  MoveL 8467 to (-32, -51.45, -12.28) mm, rotated rx 180 ry 0 rz 90 deg; joints [71.833, -17.532, 85.378, 0, 22.154, 71.833]
  MoveL 8468 to (-30.9, -50.4, -12.69) mm, rotated rx 180 ry 0 rz 90 deg; joints [71.879, -17.498, 85.311, 0, 22.187, 71.879]
  MoveL 8469 to (-30.06, -49.13, -13.09) mm, rotated rx 180 ry 0 rz 90 deg; joints [71.929, -17.47, 85.268, 0, 22.202, 71.929]
  MoveL 8470 to (-29.55, -47.71, -13.5) mm, rotated rx 180 ry 0 rz 90 deg; joints [71.98, -17.448, 85.251, 0, 22.197, 71.98]
  MoveL 8471 to (-25.22, -30.8, -13.5) mm, rotated rx 180 ry 0 rz 90 deg; joints [72.572, -17.467, 85.325, 0, 22.141, 72.572]
  MoveL 8472 to (-24.37, -27.48, -13.5) mm, rotated rx 180 ry 0 rz 90 deg; joints [72.688, -17.47, 85.338, 0, 22.131, 72.688]
  MoveL 8473 to (-24.29, -27.01, -13.5) mm, rotated rx 180 ry 0 rz 90 deg; joints [72.704, -17.471, 85.343, 0, 22.128, 72.704]
  MoveC 8474 to (-25.15, -24.96, -13.5) mm, rotated rx -180 ry 0 rz 90 deg; joints [72.762, -17.497, 85.447, 0, 22.05, 72.762] to (-27.01, -23.75, -13.5) mm, rotated rx -180 ry 0 rz 90 deg; joints [72.782, -17.536, 85.602, 0, 21.933, 72.782]
  MoveC 8475 to (-27.34, -23.73, -13.5) mm, rotated rx 180 ry 0 rz 90 deg; joints [72.78, -17.542, 85.626, 0, 21.916, 72.78] to (-27.66, -23.77, -13.5) mm, rotated rx -180 ry 0 rz 90 deg; joints [72.775, -17.547, 85.647, 0, 21.9, 72.775]
  MoveL 8476 to (-34.52, -25.11, -13.5) mm, rotated rx 180 ry 0 rz 90 deg; joints [72.662, -17.657, 86.093, 0, 21.564, 72.662]
  MoveL 8477 to (-63.97, -30.99, -13.5) mm, rotated rx 180 ry 0 rz 90 deg; joints [72.162, -18.107, 87.975, 0, 20.132, 72.162]
  MoveL 8478 to (-68.88, -32, -13.5) mm, rotated rx 180 ry 0 rz 90 deg; joints [72.076, -18.178, 88.284, 0, 19.894, 72.076]
  MoveC 8479 to (-70.35, -32.85, -13.5) mm, rotated rx -180 ry 0 rz 90 deg; joints [72.032, -18.197, 88.364, 0, 19.832, 72.032] to (-71.01, -34.41, -13.5) mm, rotated rx -180 ry 0 rz 90 deg; joints [71.974, -18.199, 88.375, 0, 19.824, 71.974]
  MoveC 8480 to (-71.02, -34.67, -13.5) mm, rotated rx -180 ry 0 rz 90 deg; joints [71.965, -18.198, 88.37, 0, 19.828, 71.965] to (-71.03, -34.93, -13.5) mm, rotated rx 180 ry 0 rz 90 deg; joints [71.956, -18.197, 88.365, 0, 19.832, 71.956]
  MoveL 8481 to (-71.03, -68.06, -13.5) mm, rotated rx 180 ry 0 rz 90 deg; joints [70.866, -18.023, 87.616, 0, 20.407, 70.866]
  MoveC 8482 to (-70.26, -69.94, -13.5) mm, rotated rx -180 ry 0 rz 90 deg; joints [70.813, -18.001, 87.521, 0, 20.48, 70.813] to (-68.4, -70.75, -13.5) mm, rotated rx 180 ry 0 rz 90 deg; joints [70.808, -17.967, 87.377, 0, 20.59, 70.808]
  MoveC 8483 to (-67.86, -70.75, -13.5) mm, rotated rx 180 ry 0 rz 90 deg; joints [70.814, -17.958, 87.34, 0, 20.618, 70.814] to (-67.31, -70.75, -13.5) mm, rotated rx 180 ry 0 rz 90 deg; joints [70.82, -17.949, 87.303, 0, 20.646, 70.82]
  MoveC 8484 to (-52.36, -70.49, -13.5) mm, rotated rx 180 ry 0 rz 90 deg; joints [70.997, -17.707, 86.295, 0, 21.412, 70.997] to (-37.4, -70.16, -13.5) mm, rotated rx 180 ry 0 rz 90 deg; joints [71.173, -17.454, 85.277, 0, 22.178, 71.173]
  MoveC 8485 to (-35.88, -69.65, -13.5) mm, rotated rx 180 ry 0 rz 90 deg; joints [71.205, -17.431, 85.183, 0, 22.248, 71.205] to (-34.9, -68.38, -13.5) mm, rotated rx 180 ry 0 rz 90 deg; joints [71.257, -17.421, 85.146, 0, 22.276, 71.257]
  MoveC 8486 to (-34.73, -67.86, -13.5) mm, rotated rx 180 ry 0 rz 90 deg; joints [71.275, -17.421, 85.146, 0, 22.276, 71.275] to (-34.59, -67.34, -13.5) mm, rotated rx 180 ry 0 rz 90 deg; joints [71.294, -17.422, 85.148, 0, 22.274, 71.294]
  MoveL 8487 to (-29.55, -47.71, -13.5) mm, rotated rx 180 ry 0 rz 90 deg; joints [71.98, -17.448, 85.251, 0, 22.197, 71.98]
  MoveL 8488 to (-36.87, -45.83, -13.5) mm, rotated rx 180 ry 0 rz 90 deg; joints [71.964, -17.585, 85.799, 0, 21.786, 71.964]
  MoveL 8489 to (-36.87, -45.83, -10.5) mm, rotated rx 180 ry 0 rz 90 deg; joints [71.964, -17.739, 85.902, 0, 21.838, 71.964]
  Establecer velocidad (1000.0 mm/s)
  MoveL 8490 to (-36.87, -45.83, 10) mm, rotated rx 180 ry 0 rz 90 deg; joints [71.964, -18.794, 86.589, 0, 22.206, 71.964]
  Establecer velocidad (66.7 mm/s)
  MoveL 8491 to (5.19, -66.61, 10) mm, rotated rx 180 ry 0 rz 90 deg; joints [71.74, -17.89, 83.159, 0, 24.731, 71.74]
  MoveL 8492 to (5.19, -66.61, -10.5) mm, rotated rx 180 ry 0 rz 90 deg; joints [71.74, -16.849, 82.47, 0, 24.38, 71.74]
  MoveL 8493 to (6.49, -67.39, -10.91) mm, rotated rx 180 ry 0 rz 90 deg; joints [71.729, -16.798, 82.344, 0, 24.454, 71.729]
  MoveL 8494 to (7.96, -67.76, -11.31) mm, rotated rx -180 ry 0 rz 90 deg; joints [71.733, -16.747, 82.216, 0, 24.531, 71.733]
  MoveL 8495 to (9.48, -67.7, -11.72) mm, rotated rx -180 ry 0 rz 90 deg; joints [71.75, -16.697, 82.094, 0, 24.602, 71.75]
  MoveL 8496 to (10.92, -67.23, -12.13) mm, rotated rx -180 ry 0 rz 90 deg; joints [71.78, -16.651, 81.988, 0, 24.663, 71.78]
  MoveL 8497 to (12.18, -66.38, -12.53) mm, rotated rx -180 ry 0 rz 90 deg; joints [71.82, -16.611, 81.903, 0, 24.708, 71.82]
  MoveL 8498 to (13.16, -65.21, -12.94) mm, rotated rx 180 ry 0 rz 90 deg; joints [71.866, -16.579, 81.847, 0, 24.732, 71.866]
  MoveL 8499 to (13.78, -63.83, -13.34) mm, rotated rx 180 ry 0 rz 90 deg; joints [71.916, -16.555, 81.821, 0, 24.734, 71.916]
  MoveL 8500 to (13.96, -62.32, -13.75) mm, rotated rx 180 ry 0 rz 90 deg; joints [71.966, -16.541, 81.829, 0, 24.711, 71.966]
  MoveL 8501 to (13.96, -51.49, -13.75) mm, rotated rx -180 ry 0 rz 90 deg; joints [72.307, -16.609, 82.081, 0, 24.528, 72.307]
  MoveL 8502 to (13.96, -34.43, -13.75) mm, rotated rx 180 ry 0 rz 90 deg; joints [72.846, -16.713, 82.466, 0, 24.247, 72.846]
  MoveC 8503 to (11.96, -34.42, -13.75) mm, rotated rx 180 ry 0 rz 90 deg; joints [72.827, -16.752, 82.61, 0, 24.141, 72.827] to (10.29, -35.54, -13.75) mm, rotated rx 180 ry 0 rz 90 deg; joints [72.775, -16.777, 82.704, 0, 24.072, 72.775]
  MoveL 8504 to (10, -36.48, -13.75) mm, rotated rx 180 ry 0 rz 90 deg; joints [72.742, -16.777, 82.705, 0, 24.072, 72.742]
  MoveL 8505 to (2.17, -64.91, -13.75) mm, rotated rx -180 ry 0 rz 90 deg; joints [71.762, -16.753, 82.614, 0, 24.139, 71.762]
  MoveL 8506 to (1.94, -65.86, -13.75) mm, rotated rx -180 ry 0 rz 90 deg; joints [71.73, -16.751, 82.608, 0, 24.143, 71.73]
  MoveC 8507 to (2.52, -67.83, -13.75) mm, rotated rx 180 ry 0 rz 90 deg; joints [71.674, -16.727, 82.52, 0, 24.207, 71.674] to (4.26, -68.91, -13.75) mm, rotated rx 180 ry 0 rz 90 deg; joints [71.658, -16.687, 82.37, 0, 24.317, 71.658]
  MoveL 8508 to (5.21, -68.93, -13.75) mm, rotated rx 180 ry 0 rz 90 deg; joints [71.667, -16.669, 82.301, 0, 24.367, 71.667]
  MoveL 8509 to (13.96, -68.54, -13.75) mm, rotated rx -180 ry 0 rz 90 deg; joints [71.77, -16.501, 81.683, 0, 24.818, 71.77]
  MoveL 8510 to (13.96, -51.49, -13.75) mm, rotated rx -180 ry 0 rz 90 deg; joints [72.307, -16.609, 82.081, 0, 24.528, 72.307]
  MoveL 8511 to (6.41, -51.49, -13.75) mm, rotated rx 180 ry 0 rz 90 deg; joints [72.23, -16.755, 82.623, 0, 24.132, 72.23]
  MoveL 8512 to (6.41, -51.49, -10.75) mm, rotated rx -180 ry 0 rz 90 deg; joints [72.23, -16.908, 82.726, 0, 24.182, 72.23]
  Establecer velocidad (1000.0 mm/s)
  MoveL 8513 to (6.41, -51.49, 10) mm, rotated rx 180 ry 0 rz 90 deg; joints [72.23, -17.962, 83.423, 0, 24.539, 72.23]
  Establecer velocidad (66.7 mm/s)
  MoveL 8514 to (-39.34, -52.07, 10) mm, rotated rx -180 ry 0 rz 90 deg; joints [71.735, -18.802, 86.618, 0, 22.184, 71.735]
  MoveL 8515 to (-39.34, -52.07, -10.5) mm, rotated rx 180 ry 0 rz 90 deg; joints [71.735, -17.747, 85.931, 0, 21.816, 71.735]
  MoveL 8516 to (-37.92, -52.63, -10.91) mm, rotated rx -180 ry 0 rz 90 deg; joints [71.732, -17.698, 85.807, 0, 21.891, 71.732]
  MoveL 8517 to (-36.42, -52.82, -11.31) mm, rotated rx -180 ry 0 rz 90 deg; joints [71.742, -17.65, 85.685, 0, 21.966, 71.742]
  MoveL 8518 to (-34.9, -52.68, -11.72) mm, rotated rx -180 ry 0 rz 90 deg; joints [71.763, -17.604, 85.57, 0, 22.035, 71.763]
  MoveL 8519 to (-33.46, -52.21, -12.13) mm, rotated rx -180 ry 0 rz 90 deg; joints [71.793, -17.561, 85.467, 0, 22.094, 71.793]
  MoveL 8520 to (-32.16, -51.43, -12.53) mm, rotated rx -180 ry 0 rz 90 deg; joints [71.832, -17.522, 85.38, 0, 22.142, 71.832]
  MoveL 8521 to (-31.06, -50.38, -12.94) mm, rotated rx -180 ry 0 rz 90 deg; joints [71.878, -17.488, 85.314, 0, 22.174, 71.878]
  MoveL 8522 to (-30.22, -49.11, -13.34) mm, rotated rx 180 ry 0 rz 90 deg; joints [71.928, -17.46, 85.271, 0, 22.189, 71.928]
  MoveL 8523 to (-29.71, -47.69, -13.75) mm, rotated rx 180 ry 0 rz 90 deg; joints [71.979, -17.438, 85.254, 0, 22.184, 71.979]
  MoveL 8524 to (-24.65, -27.96, -13.75) mm, rotated rx 180 ry 0 rz 90 deg; joints [72.67, -17.459, 85.339, 0, 22.12, 72.67]
  MoveL 8525 to (-24.53, -27.48, -13.75) mm, rotated rx -180 ry 0 rz 90 deg; joints [72.686, -17.46, 85.341, 0, 22.119, 72.686]
  MoveC 8526 to (-24.73, -26.21, -13.75) mm, rotated rx -180 ry 0 rz 90 deg; joints [72.726, -17.47, 85.383, 0, 22.088, 72.726] to (-25.42, -25.11, -13.75) mm, rotated rx -180 ry 0 rz 90 deg; joints [72.754, -17.488, 85.454, 0, 22.034, 72.754]
  MoveC 8527 to (-26.33, -24.32, -13.75) mm, rotated rx -180 ry 0 rz 90 deg; joints [72.77, -17.508, 85.535, 0, 21.974, 72.77] to (-27.48, -23.95, -13.75) mm, rotated rx 180 ry 0 rz 90 deg; joints [72.771, -17.53, 85.622, 0, 21.908, 72.771]
  MoveL 8528 to (-27.96, -24.01, -13.75) mm, rotated rx 180 ry 0 rz 90 deg; joints [72.764, -17.538, 85.654, 0, 21.884, 72.764]
  MoveL 8529 to (-31.75, -24.74, -13.75) mm, rotated rx -180 ry 0 rz 90 deg; joints [72.702, -17.599, 85.901, 0, 21.698, 72.702]
  MoveL 8530 to (-33.64, -25.11, -13.75) mm, rotated rx 180 ry 0 rz 90 deg; joints [72.671, -17.629, 86.024, 0, 21.605, 72.671]
  MoveL 8531 to (-63.97, -31.15, -13.75) mm, rotated rx 180 ry 0 rz 90 deg; joints [72.157, -18.093, 87.963, 0, 20.13, 72.157]
  MoveL 8532 to (-68.74, -32.13, -13.75) mm, rotated rx 180 ry 0 rz 90 deg; joints [72.074, -18.163, 88.264, 0, 19.899, 72.074]
  MoveC 8533 to (-70.15, -32.92, -13.75) mm, rotated rx -180 ry 0 rz 90 deg; joints [72.032, -18.18, 88.341, 0, 19.839, 72.032] to (-70.83, -34.39, -13.75) mm, rotated rx 180 ry 0 rz 90 deg; joints [71.976, -18.184, 88.355, 0, 19.829, 71.976]
  MoveC 8534 to (-70.86, -34.64, -13.75) mm, rotated rx 180 ry 0 rz 90 deg; joints [71.968, -18.183, 88.351, 0, 19.832, 71.968] to (-70.87, -34.9, -13.75) mm, rotated rx 180 ry 0 rz 90 deg; joints [71.959, -18.182, 88.346, 0, 19.836, 71.959]
  MoveL 8535 to (-70.86, -67.91, -13.75) mm, rotated rx -180 ry 0 rz 90 deg; joints [70.872, -18.008, 87.6, 0, 20.408, 70.872]
  MoveC 8536 to (-70.05, -69.85, -13.75) mm, rotated rx 180 ry 0 rz 90 deg; joints [70.818, -17.985, 87.501, 0, 20.484, 70.818] to (-68.11, -70.62, -13.75) mm, rotated rx 180 ry 0 rz 90 deg; joints [70.815, -17.95, 87.351, 0, 20.598, 70.815]
  MoveC 8537 to (-52.82, -70.34, -13.75) mm, rotated rx 180 ry 0 rz 90 deg; joints [70.996, -17.702, 86.322, 0, 21.381, 70.996] to (-37.53, -69.99, -13.75) mm, rotated rx 180 ry 0 rz 90 deg; joints [71.176, -17.445, 85.281, 0, 22.164, 71.176]
  MoveC 8538 to (-35.85, -69.39, -13.75) mm, rotated rx -180 ry 0 rz 90 deg; joints [71.214, -17.419, 85.179, 0, 22.24, 71.214] to (-34.89, -67.89, -13.75) mm, rotated rx -180 ry 0 rz 90 deg; joints [71.273, -17.411, 85.147, 0, 22.264, 71.273]
  MoveL 8539 to (-29.71, -47.69, -13.75) mm, rotated rx 180 ry 0 rz 90 deg; joints [71.979, -17.438, 85.254, 0, 22.184, 71.979]
  MoveL 8540 to (-37.02, -45.81, -13.75) mm, rotated rx 180 ry 0 rz 90 deg; joints [71.963, -17.575, 85.802, 0, 21.773, 71.963]
  MoveL 8541 to (-37.02, -45.81, -10.75) mm, rotated rx 180 ry 0 rz 90 deg; joints [71.963, -17.729, 85.904, 0, 21.825, 71.963]
  Establecer velocidad (1000.0 mm/s)
  MoveL 8542 to (-37.02, -45.81, 10) mm, rotated rx 180 ry 0 rz 90 deg; joints [71.963, -18.797, 86.6, 0, 22.197, 71.963]
  Establecer velocidad (66.7 mm/s)
  MoveL 8543 to (-62.63, 35.5, 10) mm, rotated rx 180 ry 0 rz 90 deg; joints [74.399, -19.621, 90.022, 0, 19.6, 74.399]
  MoveL 8544 to (-62.63, 35.5, -10.5) mm, rotated rx -180 ry 0 rz 90 deg; joints [74.399, -18.55, 89.334, 0, 19.216, 74.399]
  MoveL 8545 to (-64.13, 35.69, -10.91) mm, rotated rx -180 ry 0 rz 90 deg; joints [74.391, -18.552, 89.425, 0, 19.127, 74.391]
  MoveL 8546 to (-65.64, 35.51, -11.31) mm, rotated rx -180 ry 0 rz 90 deg; joints [74.371, -18.553, 89.509, 0, 19.043, 74.371]
  MoveL 8547 to (-67.07, 34.99, -11.72) mm, rotated rx 180 ry 0 rz 90 deg; joints [74.34, -18.55, 89.582, 0, 18.968, 74.34]
  MoveL 8548 to (-68.35, 34.18, -12.13) mm, rotated rx 180 ry 0 rz 90 deg; joints [74.3, -18.545, 89.639, 0, 18.906, 74.3]
  MoveL 8549 to (-69.42, 33.1, -12.53) mm, rotated rx 180 ry 0 rz 90 deg; joints [74.253, -18.535, 89.676, 0, 18.859, 74.253]
  MoveL 8550 to (-70.23, 31.81, -12.94) mm, rotated rx -180 ry 0 rz 90 deg; joints [74.202, -18.52, 89.692, 0, 18.828, 74.202]
  MoveL 8551 to (-70.73, 30.37, -13.34) mm, rotated rx -180 ry 0 rz 90 deg; joints [74.148, -18.5, 89.684, 0, 18.816, 74.148]
  MoveL 8552 to (-70.87, 28.86, -13.75) mm, rotated rx 180 ry 0 rz 90 deg; joints [74.096, -18.474, 89.651, 0, 18.824, 74.096]
  MoveL 8553 to (-70.87, 5.21, -13.75) mm, rotated rx 180 ry 0 rz 90 deg; joints [73.298, -18.372, 89.187, 0, 19.185, 73.298]
  MoveL 8554 to (-70.86, 4.4, -13.75) mm, rotated rx -180 ry 0 rz 90 deg; joints [73.27, -18.368, 89.171, 0, 19.198, 73.27]
  MoveC 8555 to (-69.84, 2.28, -13.75) mm, rotated rx -180 ry 0 rz 90 deg; joints [73.21, -18.343, 89.059, 0, 19.284, 73.21] to (-67.55, 1.73, -13.75) mm, rotated rx -180 ry 0 rz 90 deg; joints [73.214, -18.306, 88.895, 0, 19.412, 73.214]
  MoveL 8556 to (-67.28, 1.79, -13.75) mm, rotated rx -180 ry 0 rz 90 deg; joints [73.219, -18.303, 88.878, 0, 19.425, 73.219]
  MoveC 8557 to (-46.43, 6.82, -13.75) mm, rotated rx 180 ry 0 rz 90 deg; joints [73.594, -18.001, 87.567, 0, 20.433, 73.594] to (-25.61, 11.95, -13.75) mm, rotated rx 180 ry 0 rz 90 deg; joints [73.964, -17.682, 86.237, 0, 21.445, 73.964]
  MoveC 8558 to (-24.84, 12.27, -13.75) mm, rotated rx -180 ry 0 rz 90 deg; joints [73.981, -17.67, 86.19, 0, 21.48, 73.981] to (-24.21, 12.79, -13.75) mm, rotated rx -180 ry 0 rz 90 deg; joints [74.005, -17.662, 86.156, 0, 21.506, 74.005]
  MoveC 8559 to (-23.5, 14.13, -13.75) mm, rotated rx 180 ry 0 rz 90 deg; joints [74.055, -17.656, 86.133, 0, 21.523, 74.055] to (-23.5, 15.64, -13.75) mm, rotated rx -180 ry 0 rz 90 deg; joints [74.105, -17.664, 86.163, 0, 21.5, 74.105]
  MoveL 8560 to (-23.82, 16.58, -13.75) mm, rotated rx 180 ry 0 rz 90 deg; joints [74.133, -17.674, 86.204, 0, 21.469, 74.133]
  MoveL 8561 to (-28.16, 28.9, -13.75) mm, rotated rx -180 ry 0 rz 90 deg; joints [74.499, -17.805, 86.745, 0, 21.06, 74.499]
  MoveL 8562 to (-28.5, 29.83, -13.75) mm, rotated rx -180 ry 0 rz 90 deg; joints [74.527, -17.815, 86.786, 0, 21.029, 74.527]
  MoveC 8563 to (-28.94, 30.63, -13.75) mm, rotated rx 180 ry 0 rz 90 deg; joints [74.549, -17.826, 86.832, 0, 20.994, 74.549] to (-29.62, 31.24, -13.75) mm, rotated rx 180 ry 0 rz 90 deg; joints [74.564, -17.84, 86.891, 0, 20.949, 74.564]
  MoveC 8564 to (-48.19, 43.5, -13.75) mm, rotated rx -180 ry 0 rz 90 deg; joints [74.803, -18.193, 88.395, 0, 19.798, 74.803] to (-66.81, 55.67, -13.75) mm, rotated rx -180 ry 0 rz 90 deg; joints [75.046, -18.523, 89.875, 0, 18.649, 75.046]
  MoveC 8565 to (-67.27, 55.82, -13.75) mm, rotated rx 180 ry 0 rz 90 deg; joints [75.046, -18.531, 89.908, 0, 18.622, 75.046] to (-67.76, 55.86, -13.75) mm, rotated rx 180 ry 0 rz 90 deg; joints [75.043, -18.538, 89.942, 0, 18.596, 75.043]
  MoveC 8566 to (-69.28, 55.48, -13.75) mm, rotated rx 180 ry 0 rz 90 deg; joints [75.016, -18.559, 90.037, 0, 18.522, 75.016] to (-70.48, 54.47, -13.75) mm, rotated rx 180 ry 0 rz 90 deg; joints [74.971, -18.572, 90.099, 0, 18.473, 74.971]
  MoveC 8567 to (-70.77, 53.93, -13.75) mm, rotated rx -180 ry 0 rz 90 deg; joints [74.95, -18.574, 90.109, 0, 18.465, 74.95] to (-70.87, 53.33, -13.75) mm, rotated rx -180 ry 0 rz 90 deg; joints [74.929, -18.573, 90.104, 0, 18.469, 74.929]
  MoveL 8568 to (-70.87, 28.86, -13.75) mm, rotated rx 180 ry 0 rz 90 deg; joints [74.096, -18.474, 89.651, 0, 18.824, 74.096]
  MoveL 8569 to (-63.31, 28.86, -13.75) mm, rotated rx -180 ry 0 rz 90 deg; joints [74.169, -18.362, 89.144, 0, 19.218, 74.169]
  MoveL 8570 to (-63.31, 28.86, -10.75) mm, rotated rx -180 ry 0 rz 90 deg; joints [74.169, -18.519, 89.246, 0, 19.273, 74.169]
  Establecer velocidad (1000.0 mm/s)
  MoveL 8571 to (-63.31, 28.86, 10) mm, rotated rx 180 ry 0 rz 90 deg; joints [74.169, -19.603, 89.942, 0, 19.661, 74.169]
  Establecer velocidad (66.7 mm/s)
  MoveL 8572 to (13.92, 68.36, 10) mm, rotated rx -180 ry 0 rz 90 deg; joints [76.162, -18.466, 85.312, 0, 23.155, 76.162]
  MoveL 8573 to (13.92, 68.36, -10.5) mm, rotated rx 180 ry 0 rz 90 deg; joints [76.162, -17.417, 84.624, 0, 22.793, 76.162]
  MoveL 8574 to (12.79, 68.42, -10.8) mm, rotated rx -180 ry 0 rz 90 deg; joints [76.155, -17.422, 84.695, 0, 22.727, 76.155]
  MoveL 8575 to (1.8, 68.86, -13.75) mm, rotated rx 180 ry 0 rz 90 deg; joints [76.08, -17.47, 85.383, 0, 22.087, 76.08]
  MoveL 8576 to (-7.11, 69.22, -13.75) mm, rotated rx -180 ry 0 rz 90 deg; joints [76.019, -17.628, 86.017, 0, 21.611, 76.019]
  MoveL 8577 to (-10.35, 69.34, -13.75) mm, rotated rx -180 ry 0 rz 90 deg; joints [75.996, -17.684, 86.247, 0, 21.437, 75.996]
  MoveC 8578 to (-12.32, 66.93, -13.75) mm, rotated rx -180 ry 0 rz 90 deg; joints [75.9, -17.707, 86.342, 0, 21.365, 75.9] to (-12.13, 63.83, -13.75) mm, rotated rx 180 ry 0 rz 90 deg; joints [75.798, -17.691, 86.274, 0, 21.417, 75.798]
  MoveL 8579 to (-5.21, 59.19, -13.75) mm, rotated rx -180 ry 0 rz 90 deg; joints [75.703, -17.551, 85.706, 0, 21.845, 75.703]
  MoveL 8580 to (-4.12, 58.43, -13.75) mm, rotated rx 180 ry 0 rz 90 deg; joints [75.687, -17.528, 85.616, 0, 21.913, 75.687]
  MoveC 8581 to (-3.95, 58.35, -13.75) mm, rotated rx 180 ry 0 rz 90 deg; joints [75.686, -17.525, 85.602, 0, 21.923, 75.686] to (-3.77, 58.34, -13.75) mm, rotated rx 180 ry 0 rz 90 deg; joints [75.687, -17.522, 85.589, 0, 21.933, 75.687]
  MoveC 8582 to (5.1, 59.28, -13.75) mm, rotated rx 180 ry 0 rz 90 deg; joints [75.792, -17.369, 84.979, 0, 22.39, 75.792] to (13.96, 60.31, -13.75) mm, rotated rx -180 ry 0 rz 90 deg; joints [75.899, -17.213, 84.367, 0, 22.846, 75.899]
  MoveL 8583 to (13.96, 68.36, -13.75) mm, rotated rx 180 ry 0 rz 90 deg; joints [76.163, -17.249, 84.51, 0, 22.739, 76.163]
  MoveL 8584 to (12.79, 68.42, -13.75) mm, rotated rx -180 ry 0 rz 90 deg; joints [76.155, -17.271, 84.594, 0, 22.677, 76.155]
  MoveL 8585 to (1.8, 68.86, -13.75) mm, rotated rx 180 ry 0 rz 90 deg; joints [76.08, -17.47, 85.383, 0, 22.087, 76.08]
  MoveL 8586 to (1.5, 61.32, -13.75) mm, rotated rx -180 ry 0 rz 90 deg; joints [75.829, -17.442, 85.271, 0, 22.171, 75.829]
  MoveL 8587 to (1.5, 61.32, -10.75) mm, rotated rx -180 ry 0 rz 90 deg; joints [75.829, -17.597, 85.374, 0, 22.223, 75.829]
  Establecer velocidad (1000.0 mm/s)
  MoveL 8588 to (1.5, 61.32, 10) mm, rotated rx 180 ry 0 rz 90 deg; joints [75.829, -18.662, 86.069, 0, 22.593, 75.829]
  Establecer velocidad (66.7 mm/s)
  MoveL 8589 to (11.1, 65.48, 10) mm, rotated rx 180 ry 0 rz 90 deg; joints [76.045, -18.505, 85.462, 0, 23.043, 76.045]
  MoveL 8590 to (11.1, 65.48, -10.75) mm, rotated rx -180 ry 0 rz 90 deg; joints [76.045, -17.442, 84.766, 0, 22.677, 76.045]
  MoveL 8591 to (11.1, 68.29, -11.5) mm, rotated rx -180 ry 0 rz 90 deg; joints [76.137, -17.416, 84.79, 0, 22.627, 76.137]
  MoveL 8592 to (9, 68.38, -12.07) mm, rotated rx -180 ry 0 rz 90 deg; joints [76.123, -17.426, 84.921, 0, 22.505, 76.123]
  MoveL 8593 to (1.8, 68.67, -14) mm, rotated rx 180 ry 0 rz 90 deg; joints [76.074, -17.457, 85.371, 0, 22.085, 76.074]
  MoveL 8594 to (-9.74, 69.14, -14) mm, rotated rx 180 ry 0 rz 90 deg; joints [75.994, -17.66, 86.192, 0, 21.468, 75.994]
  MoveC 8595 to (-11.67, 66.75, -14) mm, rotated rx 180 ry 0 rz 90 deg; joints [75.899, -17.683, 86.285, 0, 21.397, 75.899] to (-11.49, 63.69, -14) mm, rotated rx -180 ry 0 rz 90 deg; joints [75.799, -17.666, 86.218, 0, 21.448, 75.799]
  MoveL 8596 to (-5.21, 59.48, -14) mm, rotated rx 180 ry 0 rz 90 deg; joints [75.712, -17.539, 85.703, 0, 21.836, 75.712]
  MoveL 8597 to (-4.05, 58.64, -14) mm, rotated rx -180 ry 0 rz 90 deg; joints [75.694, -17.515, 85.606, 0, 21.909, 75.694]
  MoveC 8598 to (-3.78, 58.51, -14) mm, rotated rx -180 ry 0 rz 90 deg; joints [75.693, -17.51, 85.585, 0, 21.925, 75.693] to (-3.49, 58.48, -14) mm, rotated rx 180 ry 0 rz 90 deg; joints [75.694, -17.505, 85.564, 0, 21.941, 75.694]
  MoveC 8599 to (3.81, 59.26, -14) mm, rotated rx 180 ry 0 rz 90 deg; joints [75.781, -17.379, 85.062, 0, 22.317, 75.781] to (11.1, 60.12, -14) mm, rotated rx 180 ry 0 rz 90 deg; joints [75.869, -17.251, 84.559, 0, 22.692, 75.869]
  MoveL 8600 to (11.1, 68.29, -14) mm, rotated rx 180 ry 0 rz 90 deg; joints [76.137, -17.288, 84.704, 0, 22.584, 76.137]
  MoveL 8601 to (9, 68.38, -14) mm, rotated rx -180 ry 0 rz 90 deg; joints [76.123, -17.327, 84.855, 0, 22.472, 76.123]
  MoveL 8602 to (1.8, 68.67, -14) mm, rotated rx 180 ry 0 rz 90 deg; joints [76.074, -17.457, 85.371, 0, 22.085, 76.074]
  MoveL 8603 to (1.49, 61.13, -14) mm, rotated rx -180 ry 0 rz 90 deg; joints [75.823, -17.429, 85.259, 0, 22.169, 75.823]
  MoveL 8604 to (1.49, 61.13, -11) mm, rotated rx 180 ry 0 rz 90 deg; joints [75.823, -17.583, 85.362, 0, 22.221, 75.823]
  Establecer velocidad (1000.0 mm/s)
  MoveL 8605 to (1.49, 61.13, 10) mm, rotated rx 180 ry 0 rz 90 deg; joints [75.823, -18.661, 86.066, 0, 22.595, 75.823]
  Establecer velocidad (66.7 mm/s)
  MoveL 8606 to (-62.46, 35.36, 10) mm, rotated rx 180 ry 0 rz 90 deg; joints [74.396, -19.618, 90.008, 0, 19.61, 74.396]
  MoveL 8607 to (-62.46, 35.36, -10.75) mm, rotated rx -180 ry 0 rz 90 deg; joints [74.396, -18.534, 89.312, 0, 19.222, 74.396]
  MoveL 8608 to (-63.97, 35.55, -11.16) mm, rotated rx 180 ry 0 rz 90 deg; joints [74.388, -18.536, 89.403, 0, 19.133, 74.388]
  MoveL 8609 to (-65.48, 35.37, -11.56) mm, rotated rx 180 ry 0 rz 90 deg; joints [74.368, -18.536, 89.487, 0, 19.049, 74.368]
  MoveL 8610 to (-66.91, 34.85, -11.97) mm, rotated rx 180 ry 0 rz 90 deg; joints [74.337, -18.534, 89.56, 0, 18.975, 74.337]
  MoveL 8611 to (-68.19, 34.04, -12.37) mm, rotated rx 180 ry 0 rz 90 deg; joints [74.297, -18.529, 89.617, 0, 18.912, 74.297]
  MoveL 8612 to (-69.26, 32.96, -12.78) mm, rotated rx 180 ry 0 rz 90 deg; joints [74.25, -18.519, 89.654, 0, 18.865, 74.25]
  MoveL 8613 to (-70.06, 31.67, -13.19) mm, rotated rx -180 ry 0 rz 90 deg; joints [74.199, -18.504, 89.67, 0, 18.834, 74.199]
  MoveL 8614 to (-70.56, 30.23, -13.59) mm, rotated rx 180 ry 0 rz 90 deg; joints [74.145, -18.484, 89.662, 0, 18.822, 74.145]
  MoveL 8615 to (-70.7, 28.72, -14) mm, rotated rx -180 ry 0 rz 90 deg; joints [74.093, -18.458, 89.628, 0, 18.83, 74.093]
  MoveL 8616 to (-70.7, 5.21, -14) mm, rotated rx 180 ry 0 rz 90 deg; joints [73.299, -18.356, 89.168, 0, 19.189, 73.299]
  MoveL 8617 to (-70.69, 4.26, -14) mm, rotated rx -180 ry 0 rz 90 deg; joints [73.268, -18.352, 89.148, 0, 19.204, 73.268]
  MoveC 8618 to (-70.34, 3.19, -14) mm, rotated rx 180 ry 0 rz 90 deg; joints [73.235, -18.342, 89.102, 0, 19.239, 73.235] to (-69.55, 2.37, -14) mm, rotated rx 180 ry 0 rz 90 deg; joints [73.215, -18.326, 89.033, 0, 19.293, 73.215]
  MoveC 8619 to (-68.46, 1.89, -14) mm, rotated rx 180 ry 0 rz 90 deg; joints [73.21, -18.308, 88.951, 0, 19.357, 73.21] to (-67.28, 1.94, -14) mm, rotated rx -180 ry 0 rz 90 deg; joints [73.224, -18.29, 88.872, 0, 19.418, 73.224]
  MoveC 8620 to (-46.66, 6.92, -14) mm, rotated rx 180 ry 0 rz 90 deg; joints [73.595, -17.992, 87.576, 0, 20.416, 73.595] to (-26.06, 12.01, -14) mm, rotated rx 180 ry 0 rz 90 deg; joints [73.961, -17.677, 86.261, 0, 21.416, 73.961]
  MoveL 8621 to (-25.12, 12.32, -14) mm, rotated rx 180 ry 0 rz 90 deg; joints [73.98, -17.662, 86.202, 0, 21.461, 73.98]
  MoveC 8622 to (-23.88, 13.75, -14) mm, rotated rx -180 ry 0 rz 90 deg; joints [74.039, -17.648, 86.144, 0, 21.504, 74.039] to (-23.67, 15.64, -14) mm, rotated rx 180 ry 0 rz 90 deg; joints [74.103, -17.654, 86.167, 0, 21.487, 74.103]
  MoveL 8623 to (-23.98, 16.58, -14) mm, rotated rx -180 ry 0 rz 90 deg; joints [74.131, -17.663, 86.207, 0, 21.456, 74.131]
  MoveL 8624 to (-28.32, 28.9, -14) mm, rotated rx -180 ry 0 rz 90 deg; joints [74.498, -17.795, 86.748, 0, 21.047, 74.498]
  MoveL 8625 to (-28.65, 29.78, -14) mm, rotated rx 180 ry 0 rz 90 deg; joints [74.524, -17.804, 86.787, 0, 21.017, 74.524]
  MoveC 8626 to (-29.07, 30.53, -14) mm, rotated rx 180 ry 0 rz 90 deg; joints [74.545, -17.815, 86.83, 0, 20.984, 74.545] to (-29.7, 31.1, -14) mm, rotated rx -180 ry 0 rz 90 deg; joints [74.558, -17.828, 86.885, 0, 20.943, 74.558]
  MoveC 8627 to (-48.22, 43.35, -14) mm, rotated rx 180 ry 0 rz 90 deg; joints [74.798, -18.18, 88.386, 0, 19.794, 74.798] to (-66.81, 55.51, -14) mm, rotated rx -180 ry 0 rz 90 deg; joints [75.04, -18.51, 89.863, 0, 18.646, 75.04]
  MoveC 8628 to (-68.85, 55.38, -14) mm, rotated rx 180 ry 0 rz 90 deg; joints [75.017, -18.539, 89.998, 0, 18.541, 75.017] to (-70.43, 54.09, -14) mm, rotated rx 180 ry 0 rz 90 deg; joints [74.958, -18.557, 90.08, 0, 18.476, 74.958]
  MoveC 8629 to (-70.63, 53.65, -14) mm, rotated rx 180 ry 0 rz 90 deg; joints [74.942, -18.558, 90.086, 0, 18.472, 74.942] to (-70.7, 53.18, -14) mm, rotated rx 180 ry 0 rz 90 deg; joints [74.925, -18.557, 90.082, 0, 18.475, 74.925]
  MoveL 8630 to (-70.7, 28.72, -14) mm, rotated rx -180 ry 0 rz 90 deg; joints [74.093, -18.458, 89.628, 0, 18.83, 74.093]
  MoveL 8631 to (-63.15, 28.72, -14) mm, rotated rx 180 ry 0 rz 90 deg; joints [74.165, -18.346, 89.122, 0, 19.224, 74.165]
  MoveL 8632 to (-63.15, 28.72, -11) mm, rotated rx 180 ry 0 rz 90 deg; joints [74.165, -18.503, 89.224, 0, 19.279, 74.165]
  Establecer velocidad (1000.0 mm/s)
  MoveL 8633 to (-63.15, 28.72, 10) mm, rotated rx -180 ry 0 rz 90 deg; joints [74.165, -19.6, 89.929, 0, 19.671, 74.165]
  Establecer velocidad (66.7 mm/s)
  MoveL 8634 to (-40.14, -34.96, 10) mm, rotated rx 180 ry 0 rz 90 deg; joints [72.283, -18.912, 87.056, 0, 21.856, 72.283]
  MoveL 8635 to (-40.14, -34.96, -10.75) mm, rotated rx 180 ry 0 rz 90 deg; joints [72.283, -17.842, 86.36, 0, 21.481, 72.283]
  MoveL 8636 to (-40.26, -33.45, -11.16) mm, rotated rx 180 ry 0 rz 90 deg; joints [72.331, -17.831, 86.387, 0, 21.443, 72.331]
  MoveL 8637 to (-40.73, -32, -11.56) mm, rotated rx -180 ry 0 rz 90 deg; joints [72.373, -17.825, 86.438, 0, 21.388, 72.373]
  MoveL 8638 to (-41.51, -30.7, -11.97) mm, rotated rx -180 ry 0 rz 90 deg; joints [72.408, -17.824, 86.506, 0, 21.319, 72.408]
  MoveL 8639 to (-42.56, -29.6, -12.37) mm, rotated rx 180 ry 0 rz 90 deg; joints [72.433, -17.827, 86.588, 0, 21.239, 72.433]
  MoveL 8640 to (-43.83, -28.76, -12.78) mm, rotated rx 180 ry 0 rz 90 deg; joints [72.447, -17.831, 86.679, 0, 21.152, 72.447]
  MoveL 8641 to (-45.25, -28.22, -13.19) mm, rotated rx -180 ry 0 rz 90 deg; joints [72.45, -17.836, 86.774, 0, 21.062, 72.45]
  MoveL 8642 to (-46.75, -28.01, -13.59) mm, rotated rx 180 ry 0 rz 90 deg; joints [72.441, -17.841, 86.868, 0, 20.974, 72.441]
  MoveL 8643 to (-48.26, -28.17, -14) mm, rotated rx -180 ry 0 rz 90 deg; joints [72.42, -17.844, 86.953, 0, 20.891, 72.42]
  MoveC 8644 to (-58.42, -30.2, -14) mm, rotated rx -180 ry 0 rz 90 deg; joints [72.247, -17.998, 87.601, 0, 20.397, 72.247] to (-68.59, -32.25, -14) mm, rotated rx 180 ry 0 rz 90 deg; joints [72.071, -18.147, 88.242, 0, 19.905, 72.071]
  MoveC 8645 to (-70, -33.05, -14) mm, rotated rx -180 ry 0 rz 90 deg; joints [72.03, -18.164, 88.32, 0, 19.845, 72.03] to (-70.68, -34.53, -14) mm, rotated rx -180 ry 0 rz 90 deg; joints [71.973, -18.167, 88.333, 0, 19.835, 71.973]
  MoveC 8646 to (-70.7, -34.72, -14) mm, rotated rx -180 ry 0 rz 90 deg; joints [71.967, -18.167, 88.33, 0, 19.837, 71.967] to (-70.7, -34.91, -14) mm, rotated rx -180 ry 0 rz 90 deg; joints [71.96, -18.166, 88.326, 0, 19.84, 71.96]
  MoveL 8647 to (-70.7, -67.82, -14) mm, rotated rx -180 ry 0 rz 90 deg; joints [70.877, -17.993, 87.583, 0, 20.411, 70.877]
  MoveC 8648 to (-69.9, -69.71, -14) mm, rotated rx 180 ry 0 rz 90 deg; joints [70.824, -17.97, 87.485, 0, 20.485, 70.824] to (-67.99, -70.48, -14) mm, rotated rx -180 ry 0 rz 90 deg; joints [70.821, -17.936, 87.338, 0, 20.597, 70.821]
  MoveC 8649 to (-52.79, -70.19, -14) mm, rotated rx 180 ry 0 rz 90 deg; joints [71.002, -17.69, 86.314, 0, 21.375, 71.002] to (-37.58, -69.83, -14) mm, rotated rx -180 ry 0 rz 90 deg; joints [71.181, -17.434, 85.279, 0, 22.154, 71.181]
  MoveC 8650 to (-35.95, -69.24, -14) mm, rotated rx 180 ry 0 rz 90 deg; joints [71.218, -17.409, 85.181, 0, 22.228, 71.218] to (-35.01, -67.79, -14) mm, rotated rx 180 ry 0 rz 90 deg; joints [71.275, -17.401, 85.15, 0, 22.251, 71.275]
  MoveL 8651 to (-24.81, -27.96, -14) mm, rotated rx 180 ry 0 rz 90 deg; joints [72.668, -17.449, 85.342, 0, 22.108, 72.668]
  MoveL 8652 to (-24.71, -27.48, -14) mm, rotated rx 180 ry 0 rz 90 deg; joints [72.684, -17.45, 85.345, 0, 22.105, 72.684]
  MoveC 8653 to (-25.55, -25.39, -14) mm, rotated rx 180 ry 0 rz 90 deg; joints [72.744, -17.476, 85.449, 0, 22.027, 72.744] to (-27.46, -24.17, -14) mm, rotated rx 180 ry 0 rz 90 deg; joints [72.764, -17.516, 85.607, 0, 21.908, 72.764]
  MoveC 8654 to (-27.69, -24.16, -14) mm, rotated rx -180 ry 0 rz 90 deg; joints [72.762, -17.52, 85.624, 0, 21.896, 72.762] to (-27.91, -24.18, -14) mm, rotated rx 180 ry 0 rz 90 deg; joints [72.759, -17.523, 85.639, 0, 21.885, 72.759]
  MoveC 8655 to (-38.09, -26.16, -14) mm, rotated rx -180 ry 0 rz 90 deg; joints [72.591, -17.686, 86.299, 0, 21.387, 72.591] to (-48.26, -28.17, -14) mm, rotated rx 180 ry 0 rz 90 deg; joints [72.42, -17.844, 86.953, 0, 20.891, 72.42]
  MoveL 8656 to (-46.79, -35.58, -14) mm, rotated rx -180 ry 0 rz 90 deg; joints [72.193, -17.781, 86.692, 0, 21.09, 72.193]
  MoveL 8657 to (-46.79, -35.58, -11) mm, rotated rx -180 ry 0 rz 90 deg; joints [72.193, -17.936, 86.794, 0, 21.142, 72.193]
  Establecer velocidad (1000.0 mm/s)
  MoveL 8658 to (-46.79, -35.58, 10) mm, rotated rx -180 ry 0 rz 90 deg; joints [72.193, -19.021, 87.498, 0, 21.523, 72.193]
  Establecer velocidad (66.7 mm/s)
  MoveL 8659 to (11.1, -63.95, 10) mm, rotated rx -180 ry 0 rz 90 deg; joints [71.885, -17.791, 82.798, 0, 24.993, 71.885]
  MoveL 8660 to (11.1, -63.95, -10.75) mm, rotated rx 180 ry 0 rz 90 deg; joints [71.885, -16.739, 82.1, 0, 24.639, 71.885]
  MoveL 8661 to (11.1, -51.82, -14) mm, rotated rx 180 ry 0 rz 90 deg; joints [72.267, -16.65, 82.27, 0, 24.38, 72.267]
  MoveL 8662 to (11.1, -35.18, -14) mm, rotated rx -180 ry 0 rz 90 deg; joints [72.794, -16.751, 82.646, 0, 24.105, 72.794]
  MoveC 8663 to (10.61, -35.61, -14) mm, rotated rx 180 ry 0 rz 90 deg; joints [72.776, -16.757, 82.671, 0, 24.086, 72.776] to (10.32, -36.19, -14) mm, rotated rx 180 ry 0 rz 90 deg; joints [72.755, -16.76, 82.679, 0, 24.08, 72.755]
  MoveL 8664 to (9.71, -38.38, -14) mm, rotated rx -180 ry 0 rz 90 deg; joints [72.679, -16.758, 82.674, 0, 24.084, 72.679]
  MoveL 8665 to (2.28, -65.36, -14) mm, rotated rx 180 ry 0 rz 90 deg; joints [71.749, -16.735, 82.587, 0, 24.148, 71.749]
  MoveC 8666 to (2.3, -66.77, -14) mm, rotated rx 180 ry 0 rz 90 deg; joints [71.705, -16.726, 82.552, 0, 24.173, 71.705] to (3.07, -67.94, -14) mm, rotated rx -180 ry 0 rz 90 deg; joints [71.676, -16.703, 82.469, 0, 24.234, 71.676]
  MoveC 8667 to (4.06, -68.57, -14) mm, rotated rx 180 ry 0 rz 90 deg; joints [71.667, -16.68, 82.384, 0, 24.296, 71.667] to (5.21, -68.73, -14) mm, rotated rx -180 ry 0 rz 90 deg; joints [71.673, -16.657, 82.298, 0, 24.36, 71.673]
  MoveL 8668 to (6.16, -68.68, -14) mm, rotated rx 180 ry 0 rz 90 deg; joints [71.685, -16.639, 82.231, 0, 24.408, 71.685]
  MoveL 8669 to (11.1, -68.46, -14) mm, rotated rx -180 ry 0 rz 90 deg; joints [71.743, -16.544, 81.882, 0, 24.663, 71.743]
  MoveL 8670 to (11.1, -51.82, -14) mm, rotated rx 180 ry 0 rz 90 deg; joints [72.267, -16.65, 82.27, 0, 24.38, 72.267]
  MoveL 8671 to (10.44, -44.3, -14) mm, rotated rx 180 ry 0 rz 90 deg; joints [72.499, -16.709, 82.489, 0, 24.22, 72.499]
  MoveL 8672 to (10.44, -44.3, -11) mm, rotated rx 180 ry 0 rz 90 deg; joints [72.499, -16.861, 82.592, 0, 24.27, 72.499]
  Establecer velocidad (1000.0 mm/s)
  MoveL 8673 to (10.44, -44.3, 10) mm, rotated rx 180 ry 0 rz 90 deg; joints [72.499, -17.928, 83.298, 0, 24.63, 72.499]
  Establecer velocidad (66.7 mm/s)
  MoveL 8674 to (8.24, -63.95, 10) mm, rotated rx -180 ry 0 rz 90 deg; joints [71.856, -17.847, 83.003, 0, 24.844, 71.856]
  MoveL 8675 to (8.24, -63.95, -11) mm, rotated rx 180 ry 0 rz 90 deg; joints [71.856, -16.781, 82.296, 0, 24.485, 71.856]
  MoveL 8676 to (8.24, -51.82, -14.25) mm, rotated rx -180 ry 0 rz 90 deg; joints [72.238, -16.692, 82.467, 0, 24.226, 72.238]
  MoveL 8677 to (8.24, -44.58, -14.25) mm, rotated rx 180 ry 0 rz 90 deg; joints [72.467, -16.736, 82.631, 0, 24.105, 72.467]
  MoveL 8678 to (2.63, -64.91, -14.25) mm, rotated rx 180 ry 0 rz 90 deg; joints [71.767, -16.718, 82.564, 0, 24.154, 71.767]
  MoveL 8679 to (2.47, -65.51, -14.25) mm, rotated rx -180 ry 0 rz 90 deg; joints [71.746, -16.718, 82.561, 0, 24.157, 71.746]
  MoveC 8680 to (3.18, -67.63, -14.25) mm, rotated rx -180 ry 0 rz 90 deg; joints [71.687, -16.691, 82.461, 0, 24.23, 71.687] to (5.21, -68.53, -14.25) mm, rotated rx 180 ry 0 rz 90 deg; joints [71.68, -16.646, 82.294, 0, 24.352, 71.68]
  MoveL 8681 to (8.24, -68.38, -14.25) mm, rotated rx 180 ry 0 rz 90 deg; joints [71.716, -16.588, 82.08, 0, 24.508, 71.716]
  MoveL 8682 to (8.24, -51.82, -14.25) mm, rotated rx -180 ry 0 rz 90 deg; joints [72.238, -16.692, 82.467, 0, 24.226, 72.238]
  MoveL 8683 to (8.24, -51.82, -11.25) mm, rotated rx -180 ry 0 rz 90 deg; joints [72.238, -16.845, 82.569, 0, 24.275, 72.238]
  Establecer velocidad (1000.0 mm/s)
  MoveL 8684 to (8.24, -51.82, 10) mm, rotated rx -180 ry 0 rz 90 deg; joints [72.238, -17.924, 83.284, 0, 24.64, 72.238]
  Establecer velocidad (66.7 mm/s)
  MoveL 8685 to (-39.68, -52.21, 10) mm, rotated rx 180 ry 0 rz 90 deg; joints [71.727, -18.807, 86.639, 0, 22.168, 71.727]
  MoveL 8686 to (-39.68, -52.21, -11) mm, rotated rx 180 ry 0 rz 90 deg; joints [71.727, -17.726, 85.934, 0, 21.791, 71.727]
  MoveL 8687 to (-38.27, -52.76, -11.41) mm, rotated rx 180 ry 0 rz 90 deg; joints [71.724, -17.678, 85.811, 0, 21.867, 71.724]
  MoveL 8688 to (-36.76, -52.96, -11.81) mm, rotated rx 180 ry 0 rz 90 deg; joints [71.734, -17.63, 85.688, 0, 21.941, 71.734]
  MoveL 8689 to (-35.25, -52.82, -12.22) mm, rotated rx -180 ry 0 rz 90 deg; joints [71.755, -17.584, 85.573, 0, 22.01, 71.755]
  MoveL 8690 to (-33.8, -52.35, -12.62) mm, rotated rx 180 ry 0 rz 90 deg; joints [71.785, -17.54, 85.47, 0, 22.07, 71.785]
  MoveL 8691 to (-32.5, -51.56, -13.03) mm, rotated rx -180 ry 0 rz 90 deg; joints [71.824, -17.501, 85.384, 0, 22.117, 71.824]
  MoveL 8692 to (-31.4, -50.52, -13.44) mm, rotated rx 180 ry 0 rz 90 deg; joints [71.87, -17.467, 85.318, 0, 22.15, 71.87]
  MoveL 8693 to (-30.56, -49.25, -13.84) mm, rotated rx -180 ry 0 rz 90 deg; joints [71.92, -17.439, 85.274, 0, 22.165, 71.92]
  MoveL 8694 to (-30.05, -47.82, -14.25) mm, rotated rx -180 ry 0 rz 90 deg; joints [71.971, -17.417, 85.257, 0, 22.16, 71.971]
  MoveL 8695 to (-24.98, -27.96, -14.25) mm, rotated rx -180 ry 0 rz 90 deg; joints [72.666, -17.439, 85.345, 0, 22.095, 72.666]
  MoveC 8696 to (-24.92, -27.48, -14.25) mm, rotated rx -180 ry 0 rz 90 deg; joints [72.682, -17.441, 85.351, 0, 22.09, 72.682] to (-25.01, -27.01, -14.25) mm, rotated rx 180 ry 0 rz 90 deg; joints [72.697, -17.445, 85.368, 0, 22.077, 72.697]
  MoveC 8697 to (-25.77, -25.6, -14.25) mm, rotated rx -180 ry 0 rz 90 deg; joints [72.735, -17.466, 85.451, 0, 22.015, 72.735] to (-27.01, -24.59, -14.25) mm, rotated rx 180 ry 0 rz 90 deg; joints [72.755, -17.493, 85.558, 0, 21.934, 72.755]
  MoveC 8698 to (-27.59, -24.41, -14.25) mm, rotated rx 180 ry 0 rz 90 deg; joints [72.755, -17.504, 85.603, 0, 21.901, 72.755] to (-28.2, -24.42, -14.25) mm, rotated rx -180 ry 0 rz 90 deg; joints [72.749, -17.514, 85.645, 0, 21.869, 72.749]
  MoveC 8699 to (-48.32, -28.34, -14.25) mm, rotated rx 180 ry 0 rz 90 deg; joints [72.414, -17.831, 86.945, 0, 20.886, 72.414] to (-68.42, -32.36, -14.25) mm, rotated rx -180 ry 0 rz 90 deg; joints [72.069, -18.13, 88.22, 0, 19.911, 72.069]
  MoveC 8700 to (-69.94, -33.28, -14.25) mm, rotated rx -180 ry 0 rz 90 deg; joints [72.023, -18.149, 88.302, 0, 19.847, 72.023] to (-70.54, -34.95, -14.25) mm, rotated rx -180 ry 0 rz 90 deg; joints [71.961, -18.15, 88.305, 0, 19.845, 71.961]
  MoveL 8701 to (-70.54, -66.81, -14.25) mm, rotated rx -180 ry 0 rz 90 deg; joints [70.912, -17.983, 87.587, 0, 20.397, 70.912]
  MoveL 8702 to (-70.53, -67.76, -14.25) mm, rotated rx -180 ry 0 rz 90 deg; joints [70.881, -17.978, 87.564, 0, 20.414, 70.881]
  MoveC 8703 to (-69.69, -69.63, -14.25) mm, rotated rx -180 ry 0 rz 90 deg; joints [70.83, -17.954, 87.464, 0, 20.491, 70.83] to (-67.76, -70.33, -14.25) mm, rotated rx 180 ry 0 rz 90 deg; joints [70.829, -17.92, 87.318, 0, 20.602, 70.829]
  MoveC 8704 to (-52.72, -70.03, -14.25) mm, rotated rx 180 ry 0 rz 90 deg; joints [71.007, -17.677, 86.305, 0, 21.372, 71.007] to (-37.68, -69.67, -14.25) mm, rotated rx 180 ry 0 rz 90 deg; joints [71.185, -17.423, 85.281, 0, 22.142, 71.185]
  MoveC 8705 to (-36.08, -69.09, -14.25) mm, rotated rx -180 ry 0 rz 90 deg; joints [71.221, -17.399, 85.185, 0, 22.215, 71.221] to (-35.15, -67.68, -14.25) mm, rotated rx 180 ry 0 rz 90 deg; joints [71.277, -17.391, 85.153, 0, 22.238, 71.277]
  MoveL 8706 to (-34.91, -66.81, -14.25) mm, rotated rx 180 ry 0 rz 90 deg; joints [71.307, -17.392, 85.157, 0, 22.235, 71.307]
  MoveL 8707 to (-30.05, -47.82, -14.25) mm, rotated rx -180 ry 0 rz 90 deg; joints [71.971, -17.417, 85.257, 0, 22.16, 71.971]
  MoveL 8708 to (-37.37, -45.95, -14.25) mm, rotated rx 180 ry 0 rz 90 deg; joints [71.954, -17.554, 85.805, 0, 21.749, 71.954]
  MoveL 8709 to (-37.37, -45.95, -11.25) mm, rotated rx 180 ry 0 rz 90 deg; joints [71.954, -17.709, 85.908, 0, 21.801, 71.954]
  Establecer velocidad (1000.0 mm/s)
  MoveL 8710 to (-37.37, -45.95, 10) mm, rotated rx -180 ry 0 rz 90 deg; joints [71.954, -18.802, 86.621, 0, 22.182, 71.954]
  Establecer velocidad (66.7 mm/s)
  MoveL 8711 to (-62.3, 35.47, 10) mm, rotated rx -180 ry 0 rz 90 deg; joints [74.401, -19.616, 89.999, 0, 19.617, 74.401]
  MoveL 8712 to (-62.3, 35.47, -11) mm, rotated rx -180 ry 0 rz 90 deg; joints [74.401, -18.519, 89.294, 0, 19.224, 74.401]
  MoveL 8713 to (-63.8, 35.65, -11.41) mm, rotated rx -180 ry 0 rz 90 deg; joints [74.393, -18.521, 89.385, 0, 19.135, 74.393]
  MoveL 8714 to (-65.31, 35.47, -11.81) mm, rotated rx 180 ry 0 rz 90 deg; joints [74.373, -18.521, 89.469, 0, 19.052, 74.373]
  MoveL 8715 to (-66.74, 34.96, -12.22) mm, rotated rx 180 ry 0 rz 90 deg; joints [74.342, -18.519, 89.542, 0, 18.977, 74.342]
  MoveL 8716 to (-68.02, 34.14, -12.62) mm, rotated rx 180 ry 0 rz 90 deg; joints [74.302, -18.514, 89.599, 0, 18.915, 74.302]
  MoveL 8717 to (-69.09, 33.06, -13.03) mm, rotated rx 180 ry 0 rz 90 deg; joints [74.255, -18.504, 89.636, 0, 18.867, 74.255]
  MoveL 8718 to (-69.9, 31.77, -13.44) mm, rotated rx -180 ry 0 rz 90 deg; joints [74.204, -18.489, 89.652, 0, 18.837, 74.204]
  MoveL 8719 to (-70.4, 30.34, -13.84) mm, rotated rx 180 ry 0 rz 90 deg; joints [74.15, -18.469, 89.644, 0, 18.825, 74.15]
  MoveL 8720 to (-70.54, 28.83, -14.25) mm, rotated rx 180 ry 0 rz 90 deg; joints [74.098, -18.443, 89.611, 0, 18.832, 74.098]
  MoveL 8721 to (-70.54, 4.74, -14.25) mm, rotated rx -180 ry 0 rz 90 deg; joints [73.285, -18.339, 89.139, 0, 19.2, 73.285]
  MoveC 8722 to (-69.54, 2.63, -14.25) mm, rotated rx 180 ry 0 rz 90 deg; joints [73.224, -18.314, 89.03, 0, 19.285, 73.224] to (-67.28, 2.09, -14.25) mm, rotated rx -180 ry 0 rz 90 deg; joints [73.229, -18.278, 88.867, 0, 19.411, 73.229]
  MoveC 8723 to (-46.43, 7.14, -14.25) mm, rotated rx -180 ry 0 rz 90 deg; joints [73.604, -17.976, 87.556, 0, 20.42, 73.604] to (-25.61, 12.32, -14.25) mm, rotated rx 180 ry 0 rz 90 deg; joints [73.976, -17.658, 86.227, 0, 21.431, 73.976]
  MoveC 8724 to (-24.16, 13.68, -14.25) mm, rotated rx -180 ry 0 rz 90 deg; joints [74.034, -17.64, 86.154, 0, 21.486, 74.034] to (-23.85, 15.64, -14.25) mm, rotated rx -180 ry 0 rz 90 deg; joints [74.101, -17.644, 86.171, 0, 21.473, 74.101]
  MoveL 8725 to (-24.15, 16.58, -14.25) mm, rotated rx 180 ry 0 rz 90 deg; joints [74.13, -17.653, 86.21, 0, 21.443, 74.13]
  MoveL 8726 to (-28.55, 29.07, -14.25) mm, rotated rx -180 ry 0 rz 90 deg; joints [74.501, -17.786, 86.759, 0, 21.028, 74.501]
  MoveC 8727 to (-28.66, 29.38, -14.25) mm, rotated rx 180 ry 0 rz 90 deg; joints [74.511, -17.79, 86.772, 0, 21.017, 74.511] to (-28.78, 29.7, -14.25) mm, rotated rx 180 ry 0 rz 90 deg; joints [74.52, -17.793, 86.786, 0, 21.007, 74.52]
  MoveC 8728 to (-29.19, 30.42, -14.25) mm, rotated rx 180 ry 0 rz 90 deg; joints [74.54, -17.803, 86.828, 0, 20.975, 74.54] to (-29.8, 30.98, -14.25) mm, rotated rx 180 ry 0 rz 90 deg; joints [74.553, -17.816, 86.882, 0, 20.934, 74.553]
  MoveC 8729 to (-46.9, 42.3, -14.25) mm, rotated rx 180 ry 0 rz 90 deg; joints [74.775, -18.141, 88.267, 0, 19.874, 74.775] to (-64.04, 53.54, -14.25) mm, rotated rx 180 ry 0 rz 90 deg; joints [74.998, -18.448, 89.633, 0, 18.815, 74.998]
  MoveL 8730 to (-66.33, 55.05, -14.25) mm, rotated rx 180 ry 0 rz 90 deg; joints [75.029, -18.488, 89.815, 0, 18.673, 75.029]
  MoveL 8731 to (-66.71, 55.28, -14.25) mm, rotated rx -180 ry 0 rz 90 deg; joints [75.033, -18.494, 89.844, 0, 18.65, 75.033]
  MoveC 8732 to (-68.64, 55.16, -14.25) mm, rotated rx 180 ry 0 rz 90 deg; joints [75.011, -18.522, 89.971, 0, 18.551, 75.011] to (-70.18, 53.99, -14.25) mm, rotated rx 180 ry 0 rz 90 deg; joints [74.957, -18.54, 90.053, 0, 18.486, 74.957]
  MoveC 8733 to (-70.45, 53.48, -14.25) mm, rotated rx -180 ry 0 rz 90 deg; joints [74.937, -18.541, 90.062, 0, 18.48, 74.937] to (-70.54, 52.91, -14.25) mm, rotated rx 180 ry 0 rz 90 deg; joints [74.917, -18.541, 90.058, 0, 18.483, 74.917]
  MoveL 8734 to (-70.54, 28.83, -14.25) mm, rotated rx 180 ry 0 rz 90 deg; joints [74.098, -18.443, 89.611, 0, 18.832, 74.098]
  MoveL 8735 to (-62.99, 28.83, -14.25) mm, rotated rx 180 ry 0 rz 90 deg; joints [74.17, -18.331, 89.104, 0, 19.227, 74.17]
  MoveL 8736 to (-62.99, 28.83, -11.25) mm, rotated rx -180 ry 0 rz 90 deg; joints [74.17, -18.488, 89.206, 0, 19.281, 74.17]
  Establecer velocidad (1000.0 mm/s)
  MoveL 8737 to (-62.99, 28.83, 10) mm, rotated rx 180 ry 0 rz 90 deg; joints [74.17, -19.598, 89.92, 0, 19.678, 74.17]
  Establecer velocidad (66.7 mm/s)
  MoveL 8738 to (8.24, 64.79, 10) mm, rotated rx 180 ry 0 rz 90 deg; joints [75.999, -18.555, 85.653, 0, 22.902, 75.999]
  MoveL 8739 to (8.24, 64.79, -11) mm, rotated rx 180 ry 0 rz 90 deg; joints [75.999, -17.478, 84.948, 0, 22.53, 75.999]
  MoveL 8740 to (8.24, 68.22, -11.92) mm, rotated rx -180 ry 0 rz 90 deg; joints [76.112, -17.446, 84.978, 0, 22.469, 76.112]
  MoveL 8741 to (6.16, 68.33, -12.48) mm, rotated rx -180 ry 0 rz 90 deg; joints [76.098, -17.456, 85.108, 0, 22.347, 76.098]
  MoveL 8742 to (-0.44, 68.59, -14.25) mm, rotated rx -180 ry 0 rz 90 deg; joints [76.053, -17.483, 85.52, 0, 21.963, 76.053]
  MoveL 8743 to (-9.13, 68.93, -14.25) mm, rotated rx -180 ry 0 rz 90 deg; joints [75.993, -17.636, 86.137, 0, 21.499, 75.993]
  MoveC 8744 to (-11.03, 66.57, -14.25) mm, rotated rx 180 ry 0 rz 90 deg; joints [75.899, -17.658, 86.229, 0, 21.429, 75.899] to (-10.84, 63.55, -14.25) mm, rotated rx 180 ry 0 rz 90 deg; joints [75.8, -17.642, 86.162, 0, 21.48, 75.8]
  MoveC 8745 to (-7.3, 61.18, -14.25) mm, rotated rx 180 ry 0 rz 90 deg; joints [75.751, -17.57, 85.871, 0, 21.699, 75.751] to (-3.79, 58.75, -14.25) mm, rotated rx -180 ry 0 rz 90 deg; joints [75.7, -17.498, 85.581, 0, 21.917, 75.7]
  MoveC 8746 to (-3.57, 58.63, -14.25) mm, rotated rx 180 ry 0 rz 90 deg; joints [75.698, -17.494, 85.563, 0, 21.931, 75.698] to (-3.32, 58.62, -14.25) mm, rotated rx 180 ry 0 rz 90 deg; joints [75.7, -17.489, 85.545, 0, 21.944, 75.7]
  MoveC 8747 to (2.47, 59.24, -14.25) mm, rotated rx 180 ry 0 rz 90 deg; joints [75.769, -17.39, 85.148, 0, 22.242, 75.769] to (8.24, 59.91, -14.25) mm, rotated rx 180 ry 0 rz 90 deg; joints [75.839, -17.289, 84.75, 0, 22.539, 75.839]
  MoveL 8748 to (8.24, 68.22, -14.25) mm, rotated rx 180 ry 0 rz 90 deg; joints [76.112, -17.327, 84.898, 0, 22.429, 76.112]
  MoveL 8749 to (6.16, 68.33, -14.25) mm, rotated rx -180 ry 0 rz 90 deg; joints [76.098, -17.365, 85.048, 0, 22.317, 76.098]
  MoveL 8750 to (-0.44, 68.59, -14.25) mm, rotated rx -180 ry 0 rz 90 deg; joints [76.053, -17.483, 85.52, 0, 21.963, 76.053]
  MoveL 8751 to (-0.74, 61.04, -14.25) mm, rotated rx -180 ry 0 rz 90 deg; joints [75.802, -17.455, 85.407, 0, 22.048, 75.802]
  MoveL 8752 to (-0.74, 61.04, -11.25) mm, rotated rx 180 ry 0 rz 90 deg; joints [75.802, -17.609, 85.51, 0, 22.1, 75.802]
  Establecer velocidad (1000.0 mm/s)
  MoveL 8753 to (-0.74, 61.04, 10) mm, rotated rx 180 ry 0 rz 90 deg; joints [75.802, -18.701, 86.223, 0, 22.479, 75.802]
  Establecer velocidad (66.7 mm/s)
  MoveL 8754 to (5.38, 61.88, 10) mm, rotated rx 180 ry 0 rz 90 deg; joints [75.88, -18.594, 85.804, 0, 22.79, 75.88]
  MoveL 8755 to (5.38, 61.88, -11.25) mm, rotated rx 180 ry 0 rz 90 deg; joints [75.88, -17.504, 85.091, 0, 22.413, 75.88]
  MoveL 8756 to (5.38, 68.17, -12.94) mm, rotated rx -180 ry 0 rz 90 deg; joints [76.087, -17.445, 85.145, 0, 22.301, 76.087]
  MoveL 8757 to (-0.45, 68.4, -14.5) mm, rotated rx 180 ry 0 rz 90 deg; joints [76.047, -17.469, 85.508, 0, 21.961, 76.047]
  MoveL 8758 to (-8.53, 68.73, -14.5) mm, rotated rx -180 ry 0 rz 90 deg; joints [75.991, -17.611, 86.083, 0, 21.529, 75.991]
  MoveC 8759 to (-10.39, 66.39, -14.5) mm, rotated rx 180 ry 0 rz 90 deg; joints [75.898, -17.633, 86.172, 0, 21.461, 75.898] to (-10.2, 63.4, -14.5) mm, rotated rx 180 ry 0 rz 90 deg; joints [75.801, -17.617, 86.106, 0, 21.511, 75.801]
  MoveC 8760 to (-6.87, 61.17, -14.5) mm, rotated rx 180 ry 0 rz 90 deg; joints [75.754, -17.55, 85.832, 0, 21.717, 75.754] to (-3.59, 58.86, -14.5) mm, rotated rx 180 ry 0 rz 90 deg; joints [75.706, -17.482, 85.561, 0, 21.922, 75.706]
  MoveC 8761 to (-3.39, 58.77, -14.5) mm, rotated rx 180 ry 0 rz 90 deg; joints [75.704, -17.478, 85.545, 0, 21.934, 75.704] to (-3.17, 58.75, -14.5) mm, rotated rx 180 ry 0 rz 90 deg; joints [75.706, -17.474, 85.529, 0, 21.946, 75.706]
  MoveC 8762 to (1.11, 59.21, -14.5) mm, rotated rx -180 ry 0 rz 90 deg; joints [75.757, -17.401, 85.235, 0, 22.166, 75.757] to (5.38, 59.7, -14.5) mm, rotated rx -180 ry 0 rz 90 deg; joints [75.808, -17.327, 84.941, 0, 22.386, 75.808]
  MoveL 8763 to (5.38, 68.17, -14.5) mm, rotated rx -180 ry 0 rz 90 deg; joints [76.087, -17.365, 85.091, 0, 22.274, 76.087]
  MoveL 8764 to (-0.45, 68.4, -14.5) mm, rotated rx 180 ry 0 rz 90 deg; joints [76.047, -17.469, 85.508, 0, 21.961, 76.047]
  MoveL 8765 to (-0.75, 60.86, -14.5) mm, rotated rx -180 ry 0 rz 90 deg; joints [75.795, -17.441, 85.396, 0, 22.045, 75.795]
  MoveL 8766 to (-0.75, 60.86, -11.5) mm, rotated rx 180 ry 0 rz 90 deg; joints [75.795, -17.596, 85.499, 0, 22.097, 75.795]
  Establecer velocidad (1000.0 mm/s)
  MoveL 8767 to (-0.75, 60.86, 10) mm, rotated rx 180 ry 0 rz 90 deg; joints [75.795, -18.701, 86.22, 0, 22.48, 75.795]
  Establecer velocidad (66.7 mm/s)
  MoveL 8768 to (-62.13, 35.52, 10) mm, rotated rx 180 ry 0 rz 90 deg; joints [74.404, -19.614, 89.989, 0, 19.625, 74.404]
  MoveL 8769 to (-62.13, 35.52, -11.25) mm, rotated rx 180 ry 0 rz 90 deg; joints [74.404, -18.503, 89.276, 0, 19.228, 74.404]
  MoveL 8770 to (-63.64, 35.7, -11.66) mm, rotated rx 180 ry 0 rz 90 deg; joints [74.397, -18.505, 89.367, 0, 19.139, 74.397]
  MoveL 8771 to (-65.15, 35.52, -12.06) mm, rotated rx 180 ry 0 rz 90 deg; joints [74.376, -18.506, 89.451, 0, 19.055, 74.376]
  MoveL 8772 to (-66.58, 35.01, -12.47) mm, rotated rx 180 ry 0 rz 90 deg; joints [74.345, -18.504, 89.524, 0, 18.98, 74.345]
  MoveL 8773 to (-67.86, 34.19, -12.88) mm, rotated rx 180 ry 0 rz 90 deg; joints [74.305, -18.498, 89.58, 0, 18.918, 74.305]
  MoveL 8774 to (-68.93, 33.11, -13.28) mm, rotated rx -180 ry 0 rz 90 deg; joints [74.259, -18.488, 89.618, 0, 18.87, 74.259]
  MoveL 8775 to (-69.73, 31.82, -13.69) mm, rotated rx -180 ry 0 rz 90 deg; joints [74.207, -18.473, 89.633, 0, 18.84, 74.207]
  MoveL 8776 to (-70.23, 30.39, -14.09) mm, rotated rx 180 ry 0 rz 90 deg; joints [74.154, -18.453, 89.626, 0, 18.828, 74.154]
  MoveL 8777 to (-70.37, 28.88, -14.5) mm, rotated rx -180 ry 0 rz 90 deg; joints [74.101, -18.428, 89.592, 0, 18.836, 74.101]
  MoveL 8778 to (-70.37, 4.88, -14.5) mm, rotated rx 180 ry 0 rz 90 deg; joints [73.291, -18.324, 89.122, 0, 19.202, 73.291]
  MoveC 8779 to (-69.35, 2.78, -14.5) mm, rotated rx -180 ry 0 rz 90 deg; joints [73.231, -18.299, 89.011, 0, 19.288, 73.231] to (-67.07, 2.28, -14.5) mm, rotated rx 180 ry 0 rz 90 deg; joints [73.237, -18.262, 88.848, 0, 19.414, 73.237]
  MoveC 8780 to (-46.55, 7.26, -14.5) mm, rotated rx 180 ry 0 rz 90 deg; joints [73.607, -17.966, 87.559, 0, 20.407, 73.607] to (-26.06, 12.37, -14.5) mm, rotated rx 180 ry 0 rz 90 deg; joints [73.973, -17.652, 86.251, 0, 21.402, 73.973]
  MoveC 8781 to (-25.08, 12.87, -14.5) mm, rotated rx -180 ry 0 rz 90 deg; joints [73.999, -17.638, 86.193, 0, 21.445, 73.999] to (-24.41, 13.74, -14.5) mm, rotated rx -180 ry 0 rz 90 deg; joints [74.034, -17.631, 86.163, 0, 21.468, 74.034]
  MoveC 8782 to (-24.01, 14.92, -14.5) mm, rotated rx 180 ry 0 rz 90 deg; joints [74.076, -17.63, 86.159, 0, 21.471, 74.076] to (-24.17, 16.15, -14.5) mm, rotated rx 180 ry 0 rz 90 deg; joints [74.115, -17.639, 86.194, 0, 21.444, 74.115]
  MoveL 8783 to (-28.64, 28.9, -14.5) mm, rotated rx 180 ry 0 rz 90 deg; joints [74.495, -17.774, 86.753, 0, 21.021, 74.495]
  MoveL 8784 to (-28.9, 29.6, -14.5) mm, rotated rx -180 ry 0 rz 90 deg; joints [74.516, -17.782, 86.784, 0, 20.997, 74.516]
  MoveC 8785 to (-29.29, 30.28, -14.5) mm, rotated rx 180 ry 0 rz 90 deg; joints [74.535, -17.791, 86.824, 0, 20.967, 74.535] to (-29.85, 30.82, -14.5) mm, rotated rx 180 ry 0 rz 90 deg; joints [74.547, -17.803, 86.873, 0, 20.93, 74.547]
  MoveC 8786 to (-48.18, 42.98, -14.5) mm, rotated rx -180 ry 0 rz 90 deg; joints [74.786, -18.151, 88.359, 0, 19.793, 74.786] to (-66.58, 55.03, -14.5) mm, rotated rx -180 ry 0 rz 90 deg; joints [75.026, -18.478, 89.822, 0, 18.656, 75.026]
  MoveC 8787 to (-68.61, 54.86, -14.5) mm, rotated rx -180 ry 0 rz 90 deg; joints [75.001, -18.507, 89.955, 0, 18.552, 75.001] to (-70.16, 53.54, -14.5) mm, rotated rx -180 ry 0 rz 90 deg; joints [74.942, -18.524, 90.035, 0, 18.489, 74.942]
  MoveC 8788 to (-70.31, 53.23, -14.5) mm, rotated rx 180 ry 0 rz 90 deg; joints [74.93, -18.525, 90.04, 0, 18.486, 74.93] to (-70.37, 52.88, -14.5) mm, rotated rx 180 ry 0 rz 90 deg; joints [74.918, -18.525, 90.038, 0, 18.487, 74.918]
  MoveL 8789 to (-70.37, 28.88, -14.5) mm, rotated rx -180 ry 0 rz 90 deg; joints [74.101, -18.428, 89.592, 0, 18.836, 74.101]
  MoveL 8790 to (-62.82, 28.88, -14.5) mm, rotated rx 180 ry 0 rz 90 deg; joints [74.174, -18.316, 89.085, 0, 19.23, 74.174]
  MoveL 8791 to (-62.82, 28.88, -11.5) mm, rotated rx 180 ry 0 rz 90 deg; joints [74.174, -18.472, 89.188, 0, 19.285, 74.174]
  Establecer velocidad (1000.0 mm/s)
  MoveL 8792 to (-62.82, 28.88, 10) mm, rotated rx -180 ry 0 rz 90 deg; joints [74.174, -19.596, 89.909, 0, 19.686, 74.174]
  Establecer velocidad (66.7 mm/s)
  MoveL 8793 to (-40, -35.27, 10) mm, rotated rx 180 ry 0 rz 90 deg; joints [72.274, -18.908, 87.039, 0, 21.868, 72.274]
  MoveL 8794 to (-40, -35.27, -11.25) mm, rotated rx -180 ry 0 rz 90 deg; joints [72.274, -17.812, 86.327, 0, 21.485, 72.274]
  MoveL 8795 to (-40.11, -33.75, -11.66) mm, rotated rx -180 ry 0 rz 90 deg; joints [72.322, -17.801, 86.353, 0, 21.447, 72.322]
  MoveL 8796 to (-40.58, -32.31, -12.06) mm, rotated rx 180 ry 0 rz 90 deg; joints [72.365, -17.795, 86.404, 0, 21.392, 72.365]
  MoveL 8797 to (-41.36, -31, -12.47) mm, rotated rx 180 ry 0 rz 90 deg; joints [72.399, -17.794, 86.472, 0, 21.323, 72.399]
  MoveL 8798 to (-42.41, -29.9, -12.88) mm, rotated rx 180 ry 0 rz 90 deg; joints [72.424, -17.797, 86.554, 0, 21.243, 72.424]
  MoveL 8799 to (-43.67, -29.06, -13.28) mm, rotated rx -180 ry 0 rz 90 deg; joints [72.439, -17.801, 86.645, 0, 21.156, 72.439]
  MoveL 8800 to (-45.1, -28.52, -13.69) mm, rotated rx 180 ry 0 rz 90 deg; joints [72.442, -17.806, 86.74, 0, 21.066, 72.442]
  MoveL 8801 to (-46.6, -28.31, -14.09) mm, rotated rx -180 ry 0 rz 90 deg; joints [72.433, -17.811, 86.834, 0, 20.978, 72.433]
  MoveL 8802 to (-48.11, -28.47, -14.5) mm, rotated rx 180 ry 0 rz 90 deg; joints [72.412, -17.814, 86.919, 0, 20.895, 72.412]
  MoveC 8803 to (-58.17, -30.46, -14.5) mm, rotated rx 180 ry 0 rz 90 deg; joints [72.241, -17.966, 87.561, 0, 20.405, 72.241] to (-68.23, -32.48, -14.5) mm, rotated rx 180 ry 0 rz 90 deg; joints [72.067, -18.114, 88.196, 0, 19.918, 72.067]
  MoveC 8804 to (-69.77, -33.38, -14.5) mm, rotated rx 180 ry 0 rz 90 deg; joints [72.021, -18.133, 88.28, 0, 19.853, 72.021] to (-70.37, -35.06, -14.5) mm, rotated rx 180 ry 0 rz 90 deg; joints [71.959, -18.134, 88.283, 0, 19.851, 71.959]
  MoveL 8805 to (-70.37, -35.54, -14.5) mm, rotated rx -180 ry 0 rz 90 deg; joints [71.943, -18.132, 88.273, 0, 19.859, 71.943]
  MoveL 8806 to (-70.37, -66.81, -14.5) mm, rotated rx -180 ry 0 rz 90 deg; joints [70.914, -17.968, 87.567, 0, 20.401, 70.914]
  MoveL 8807 to (-70.35, -67.63, -14.5) mm, rotated rx -180 ry 0 rz 90 deg; joints [70.887, -17.963, 87.547, 0, 20.416, 70.887]
  MoveC 8808 to (-69.56, -69.45, -14.5) mm, rotated rx -180 ry 0 rz 90 deg; joints [70.837, -17.94, 87.451, 0, 20.49, 70.837] to (-67.71, -70.18, -14.5) mm, rotated rx -180 ry 0 rz 90 deg; joints [70.834, -17.907, 87.309, 0, 20.597, 70.834]
  MoveL 8809 to (-66.81, -70.17, -14.5) mm, rotated rx 180 ry 0 rz 90 deg; joints [70.845, -17.893, 87.249, 0, 20.644, 70.845]
  MoveL 8810 to (-42.99, -69.65, -14.5) mm, rotated rx 180 ry 0 rz 90 deg; joints [71.127, -17.502, 85.639, 0, 21.863, 71.127]
  MoveL 8811 to (-37.79, -69.51, -14.5) mm, rotated rx -180 ry 0 rz 90 deg; joints [71.189, -17.413, 85.284, 0, 22.129, 71.189]
  MoveC 8812 to (-36.22, -68.96, -14.5) mm, rotated rx 180 ry 0 rz 90 deg; joints [71.224, -17.389, 85.189, 0, 22.201, 71.224] to (-35.28, -67.58, -14.5) mm, rotated rx 180 ry 0 rz 90 deg; joints [71.279, -17.381, 85.156, 0, 22.225, 71.279]
  MoveC 8813 to (-35.08, -66.88, -14.5) mm, rotated rx 180 ry 0 rz 90 deg; joints [71.303, -17.382, 85.159, 0, 22.223, 71.303] to (-34.9, -66.18, -14.5) mm, rotated rx -180 ry 0 rz 90 deg; joints [71.328, -17.383, 85.163, 0, 22.22, 71.328]
  MoveL 8814 to (-25.14, -27.96, -14.5) mm, rotated rx 180 ry 0 rz 90 deg; joints [72.665, -17.429, 85.347, 0, 22.082, 72.665]
  MoveC 8815 to (-25.37, -26.74, -14.5) mm, rotated rx 180 ry 0 rz 90 deg; joints [72.702, -17.44, 85.39, 0, 22.05, 72.702] to (-26.06, -25.71, -14.5) mm, rotated rx -180 ry 0 rz 90 deg; joints [72.728, -17.457, 85.46, 0, 21.997, 72.728]
  MoveC 8816 to (-26.91, -24.98, -14.5) mm, rotated rx 180 ry 0 rz 90 deg; joints [72.743, -17.476, 85.535, 0, 21.941, 72.743] to (-27.96, -24.59, -14.5) mm, rotated rx -180 ry 0 rz 90 deg; joints [72.746, -17.496, 85.616, 0, 21.88, 72.746]
  MoveL 8817 to (-28.43, -24.65, -14.5) mm, rotated rx 180 ry 0 rz 90 deg; joints [72.739, -17.504, 85.647, 0, 21.857, 72.739]
  MoveL 8818 to (-30.8, -25.09, -14.5) mm, rotated rx -180 ry 0 rz 90 deg; joints [72.701, -17.542, 85.802, 0, 21.74, 72.701]
  MoveC 8819 to (-39.45, -26.77, -14.5) mm, rotated rx 180 ry 0 rz 90 deg; joints [72.557, -17.68, 86.363, 0, 21.317, 72.557] to (-48.11, -28.47, -14.5) mm, rotated rx -180 ry 0 rz 90 deg; joints [72.412, -17.814, 86.919, 0, 20.895, 72.412]
  MoveL 8820 to (-46.65, -35.87, -14.5) mm, rotated rx -180 ry 0 rz 90 deg; joints [72.185, -17.751, 86.658, 0, 21.093, 72.185]
  MoveL 8821 to (-46.65, -35.87, -11.5) mm, rotated rx 180 ry 0 rz 90 deg; joints [72.185, -17.906, 86.761, 0, 21.146, 72.185]
  Establecer velocidad (1000.0 mm/s)
  MoveL 8822 to (-46.65, -35.87, 10) mm, rotated rx 180 ry 0 rz 90 deg; joints [72.185, -19.017, 87.482, 0, 21.536, 72.185]
  Establecer velocidad (66.7 mm/s)
  MoveL 8823 to (3.1, -64.02, 10) mm, rotated rx -180 ry 0 rz 90 deg; joints [71.8, -17.947, 83.369, 0, 24.579, 71.8]
  MoveL 8824 to (3.1, -64.02, -11.25) mm, rotated rx 180 ry 0 rz 90 deg; joints [71.8, -16.868, 82.654, 0, 24.214, 71.8]
  MoveL 8825 to (2.85, -64.91, -11.5) mm, rotated rx 180 ry 0 rz 90 deg; joints [71.769, -16.854, 82.642, 0, 24.212, 71.769]
  MoveL 8826 to (2.72, -65.53, -11.67) mm, rotated rx 180 ry 0 rz 90 deg; joints [71.748, -16.844, 82.631, 0, 24.213, 71.748]
  MoveL 8827 to (2.73, -65.95, -11.78) mm, rotated rx -180 ry 0 rz 90 deg; joints [71.735, -16.836, 82.617, 0, 24.218, 71.735]
  MoveL 8828 to (3.13, -67.02, -12.09) mm, rotated rx -180 ry 0 rz 90 deg; joints [71.706, -16.805, 82.553, 0, 24.253, 71.706]
  MoveL 8829 to (3.92, -67.86, -12.4) mm, rotated rx -180 ry 0 rz 90 deg; joints [71.688, -16.769, 82.466, 0, 24.303, 71.688]
  MoveL 8830 to (4.97, -68.31, -12.7) mm, rotated rx -180 ry 0 rz 90 deg; joints [71.684, -16.73, 82.369, 0, 24.361, 71.684]
  MoveL 8831 to (5.38, -68.34, -12.81) mm, rotated rx 180 ry 0 rz 90 deg; joints [71.688, -16.717, 82.335, 0, 24.381, 71.688]
  MoveL 8832 to (5.38, -62.04, -14.5) mm, rotated rx 180 ry 0 rz 90 deg; joints [71.886, -16.671, 82.426, 0, 24.245, 71.886]
  MoveL 8833 to (5.38, -55.75, -14.5) mm, rotated rx 180 ry 0 rz 90 deg; joints [72.085, -16.71, 82.572, 0, 24.138, 72.085]
  MoveL 8834 to (2.85, -64.91, -14.5) mm, rotated rx -180 ry 0 rz 90 deg; joints [71.769, -16.701, 82.539, 0, 24.162, 71.769]
  MoveL 8835 to (2.72, -65.53, -14.5) mm, rotated rx 180 ry 0 rz 90 deg; joints [71.748, -16.7, 82.534, 0, 24.166, 71.748]
  MoveC 8836 to (3.5, -67.46, -14.5) mm, rotated rx -180 ry 0 rz 90 deg; joints [71.696, -16.673, 82.433, 0, 24.24, 71.696] to (5.38, -68.34, -14.5) mm, rotated rx -180 ry 0 rz 90 deg; joints [71.688, -16.631, 82.277, 0, 24.353, 71.688]
  MoveL 8837 to (5.38, -62.04, -14.5) mm, rotated rx 180 ry 0 rz 90 deg; joints [71.886, -16.671, 82.426, 0, 24.245, 71.886]
  MoveL 8838 to (5.38, -62.04, -11.5) mm, rotated rx 180 ry 0 rz 90 deg; joints [71.886, -16.823, 82.529, 0, 24.295, 71.886]
  Establecer velocidad (1000.0 mm/s)
  MoveL 8839 to (5.38, -62.04, 10) mm, rotated rx 180 ry 0 rz 90 deg; joints [71.886, -17.915, 83.252, 0, 24.663, 71.886]
  Establecer velocidad (66.7 mm/s)
  MoveL 8840 to (-40.03, -52.35, 10) mm, rotated rx -180 ry 0 rz 90 deg; joints [71.719, -18.812, 86.659, 0, 22.153, 71.719]
  MoveL 8841 to (-40.03, -52.35, -11.5) mm, rotated rx -180 ry 0 rz 90 deg; joints [71.719, -17.705, 85.938, 0, 21.767, 71.719]
  MoveL 8842 to (-38.61, -52.9, -11.91) mm, rotated rx 180 ry 0 rz 90 deg; joints [71.716, -17.657, 85.814, 0, 21.843, 71.716]
  MoveL 8843 to (-37.11, -53.09, -12.31) mm, rotated rx 180 ry 0 rz 90 deg; joints [71.726, -17.609, 85.692, 0, 21.917, 71.726]
  MoveL 8844 to (-35.59, -52.95, -12.72) mm, rotated rx -180 ry 0 rz 90 deg; joints [71.747, -17.563, 85.577, 0, 21.986, 71.747]
  MoveL 8845 to (-34.15, -52.48, -13.12) mm, rotated rx 180 ry 0 rz 90 deg; joints [71.777, -17.52, 85.474, 0, 22.046, 71.777]
  MoveL 8846 to (-32.84, -51.7, -13.53) mm, rotated rx 180 ry 0 rz 90 deg; joints [71.816, -17.481, 85.388, 0, 22.093, 71.816]
  MoveL 8847 to (-31.75, -50.65, -13.94) mm, rotated rx -180 ry 0 rz 90 deg; joints [71.862, -17.447, 85.321, 0, 22.125, 71.862]
  MoveL 8848 to (-30.91, -49.38, -14.34) mm, rotated rx -180 ry 0 rz 90 deg; joints [71.912, -17.419, 85.278, 0, 22.14, 71.912]
  MoveL 8849 to (-30.4, -47.95, -14.75) mm, rotated rx -180 ry 0 rz 90 deg; joints [71.963, -17.397, 85.261, 0, 22.136, 71.963]
  MoveL 8850 to (-25.42, -28.43, -14.75) mm, rotated rx 180 ry 0 rz 90 deg; joints [72.646, -17.419, 85.348, 0, 22.071, 72.646]
  MoveL 8851 to (-25.33, -28.05, -14.75) mm, rotated rx 180 ry 0 rz 90 deg; joints [72.66, -17.419, 85.35, 0, 22.069, 72.66]
  MoveC 8852 to (-26.15, -26.03, -14.75) mm, rotated rx 180 ry 0 rz 90 deg; joints [72.717, -17.444, 85.45, 0, 21.994, 72.717] to (-27.96, -24.83, -14.75) mm, rotated rx -180 ry 0 rz 90 deg; joints [72.738, -17.482, 85.602, 0, 21.88, 72.738]
  MoveC 8853 to (-28.44, -24.84, -14.75) mm, rotated rx -180 ry 0 rz 90 deg; joints [72.732, -17.49, 85.635, 0, 21.855, 72.732] to (-28.91, -24.91, -14.75) mm, rotated rx 180 ry 0 rz 90 deg; joints [72.725, -17.498, 85.667, 0, 21.831, 72.725]
  MoveC 8854 to (-48.53, -28.71, -14.75) mm, rotated rx -180 ry 0 rz 90 deg; joints [72.4, -17.807, 86.935, 0, 20.872, 72.4] to (-68.14, -32.61, -14.75) mm, rotated rx -180 ry 0 rz 90 deg; joints [72.064, -18.099, 88.178, 0, 19.92, 72.064]
  MoveC 8855 to (-69.62, -33.5, -14.75) mm, rotated rx 180 ry 0 rz 90 deg; joints [72.019, -18.117, 88.259, 0, 19.859, 72.019] to (-70.21, -35.13, -14.75) mm, rotated rx 180 ry 0 rz 90 deg; joints [71.958, -18.118, 88.262, 0, 19.856, 71.958]
  MoveL 8856 to (-70.21, -67.24, -14.75) mm, rotated rx 180 ry 0 rz 90 deg; joints [70.902, -17.95, 87.537, 0, 20.412, 70.902]
  MoveC 8857 to (-70.19, -67.59, -14.75) mm, rotated rx 180 ry 0 rz 90 deg; joints [70.89, -17.948, 87.528, 0, 20.419, 70.89] to (-70.14, -67.93, -14.75) mm, rotated rx 180 ry 0 rz 90 deg; joints [70.88, -17.945, 87.517, 0, 20.428, 70.88]
  MoveC 8858 to (-69.25, -69.44, -14.75) mm, rotated rx -180 ry 0 rz 90 deg; joints [70.84, -17.923, 87.422, 0, 20.501, 70.84] to (-67.6, -70.02, -14.75) mm, rotated rx -180 ry 0 rz 90 deg; joints [70.84, -17.893, 87.297, 0, 20.596, 70.84]
  MoveL 8859 to (-63.97, -69.96, -14.75) mm, rotated rx 180 ry 0 rz 90 deg; joints [70.883, -17.835, 87.053, 0, 20.782, 70.883]
  MoveL 8860 to (-39.33, -69.4, -14.75) mm, rotated rx -180 ry 0 rz 90 deg; joints [71.176, -17.428, 85.384, 0, 22.043, 71.176]
  MoveL 8861 to (-37.91, -69.35, -14.75) mm, rotated rx 180 ry 0 rz 90 deg; joints [71.193, -17.404, 85.287, 0, 22.116, 71.193]
  MoveC 8862 to (-36.47, -68.9, -14.75) mm, rotated rx 180 ry 0 rz 90 deg; joints [71.223, -17.381, 85.199, 0, 22.182, 71.223] to (-35.5, -67.76, -14.75) mm, rotated rx -180 ry 0 rz 90 deg; joints [71.27, -17.371, 85.159, 0, 22.213, 71.27]
  MoveL 8863 to (-35.21, -66.81, -14.75) mm, rotated rx 180 ry 0 rz 90 deg; joints [71.304, -17.372, 85.161, 0, 22.211, 71.304]
  MoveL 8864 to (-30.4, -47.95, -14.75) mm, rotated rx -180 ry 0 rz 90 deg; joints [71.963, -17.397, 85.261, 0, 22.136, 71.963]
  MoveL 8865 to (-37.72, -46.08, -14.75) mm, rotated rx -180 ry 0 rz 90 deg; joints [71.946, -17.533, 85.809, 0, 21.724, 71.946]
  MoveL 8866 to (-37.72, -46.08, -11.75) mm, rotated rx -180 ry 0 rz 90 deg; joints [71.946, -17.688, 85.912, 0, 21.776, 71.946]
  Establecer velocidad (1000.0 mm/s)
  MoveL 8867 to (-37.72, -46.08, 10) mm, rotated rx 180 ry 0 rz 90 deg; joints [71.946, -18.808, 86.642, 0, 22.166, 71.946]
  Establecer velocidad (66.7 mm/s)
  MoveL 8868 to (-61.97, 35.24, 10) mm, rotated rx 180 ry 0 rz 90 deg; joints [74.397, -19.61, 89.973, 0, 19.638, 74.397]
  MoveL 8869 to (-61.97, 35.24, -11.5) mm, rotated rx -180 ry 0 rz 90 deg; joints [74.397, -18.487, 89.251, 0, 19.236, 74.397]
  MoveL 8870 to (-63.47, 35.42, -11.91) mm, rotated rx 180 ry 0 rz 90 deg; joints [74.389, -18.489, 89.342, 0, 19.147, 74.389]
  MoveL 8871 to (-64.98, 35.24, -12.31) mm, rotated rx 180 ry 0 rz 90 deg; joints [74.368, -18.489, 89.426, 0, 19.063, 74.368]
  MoveL 8872 to (-66.41, 34.73, -12.72) mm, rotated rx -180 ry 0 rz 90 deg; joints [74.337, -18.487, 89.499, 0, 18.989, 74.337]
  MoveL 8873 to (-67.7, 33.91, -13.12) mm, rotated rx -180 ry 0 rz 90 deg; joints [74.297, -18.482, 89.555, 0, 18.926, 74.297]
  MoveL 8874 to (-68.77, 32.83, -13.53) mm, rotated rx 180 ry 0 rz 90 deg; joints [74.251, -18.472, 89.593, 0, 18.879, 74.251]
  MoveL 8875 to (-69.57, 31.54, -13.94) mm, rotated rx 180 ry 0 rz 90 deg; joints [74.199, -18.457, 89.608, 0, 18.848, 74.199]
  MoveL 8876 to (-70.07, 30.11, -14.34) mm, rotated rx 180 ry 0 rz 90 deg; joints [74.146, -18.437, 89.601, 0, 18.836, 74.146]
  MoveL 8877 to (-70.21, 28.6, -14.75) mm, rotated rx 180 ry 0 rz 90 deg; joints [74.093, -18.411, 89.567, 0, 18.844, 74.093]
  MoveL 8878 to (-70.21, 5.21, -14.75) mm, rotated rx -180 ry 0 rz 90 deg; joints [73.304, -18.31, 89.109, 0, 19.201, 73.304]
  MoveL 8879 to (-70.2, 4.74, -14.75) mm, rotated rx 180 ry 0 rz 90 deg; joints [73.288, -18.307, 89.099, 0, 19.209, 73.288]
  MoveC 8880 to (-69.03, 2.83, -14.75) mm, rotated rx 180 ry 0 rz 90 deg; joints [73.236, -18.281, 88.982, 0, 19.3, 73.236] to (-66.81, 2.48, -14.75) mm, rotated rx 180 ry 0 rz 90 deg; joints [73.247, -18.246, 88.826, 0, 19.42, 73.247]
  MoveC 8881 to (-46.56, 7.42, -14.75) mm, rotated rx 180 ry 0 rz 90 deg; joints [73.613, -17.954, 87.554, 0, 20.4, 73.613] to (-26.33, 12.47, -14.75) mm, rotated rx -180 ry 0 rz 90 deg; joints [73.974, -17.645, 86.263, 0, 21.381, 73.974]
  MoveC 8882 to (-25.93, 12.6, -14.75) mm, rotated rx -180 ry 0 rz 90 deg; joints [73.982, -17.639, 86.238, 0, 21.401, 73.982] to (-25.54, 12.79, -14.75) mm, rotated rx 180 ry 0 rz 90 deg; joints [73.992, -17.633, 86.215, 0, 21.418, 73.992]
  MoveC 8883 to (-24.51, 14.04, -14.75) mm, rotated rx 180 ry 0 rz 90 deg; joints [74.043, -17.621, 86.168, 0, 21.454, 74.043] to (-24.2, 15.64, -14.75) mm, rotated rx 180 ry 0 rz 90 deg; joints [74.098, -17.624, 86.178, 0, 21.446, 74.098]
  MoveL 8884 to (-24.33, 16.11, -14.75) mm, rotated rx 180 ry 0 rz 90 deg; joints [74.113, -17.628, 86.196, 0, 21.432, 74.113]
  MoveL 8885 to (-24.49, 16.58, -14.75) mm, rotated rx 180 ry 0 rz 90 deg; joints [74.127, -17.633, 86.216, 0, 21.417, 74.127]
  MoveL 8886 to (-28.97, 29.35, -14.75) mm, rotated rx -180 ry 0 rz 90 deg; joints [74.507, -17.769, 86.775, 0, 20.993, 74.507]
  MoveC 8887 to (-29.4, 30.15, -14.75) mm, rotated rx 180 ry 0 rz 90 deg; joints [74.529, -17.78, 86.821, 0, 20.959, 74.529] to (-30.07, 30.77, -14.75) mm, rotated rx 180 ry 0 rz 90 deg; joints [74.544, -17.793, 86.878, 0, 20.915, 74.544]
  MoveC 8888 to (-48.23, 42.83, -14.75) mm, rotated rx -180 ry 0 rz 90 deg; joints [74.78, -18.138, 88.351, 0, 19.788, 74.78] to (-66.45, 54.79, -14.75) mm, rotated rx -180 ry 0 rz 90 deg; joints [75.019, -18.462, 89.801, 0, 18.662, 75.019]
  MoveC 8889 to (-68.35, 54.67, -14.75) mm, rotated rx -180 ry 0 rz 90 deg; joints [74.997, -18.489, 89.926, 0, 18.564, 74.997] to (-69.86, 53.52, -14.75) mm, rotated rx 180 ry 0 rz 90 deg; joints [74.944, -18.507, 90.006, 0, 18.501, 74.944]
  MoveC 8890 to (-70.12, 53.02, -14.75) mm, rotated rx 180 ry 0 rz 90 deg; joints [74.925, -18.509, 90.014, 0, 18.494, 74.925] to (-70.21, 52.46, -14.75) mm, rotated rx -180 ry 0 rz 90 deg; joints [74.905, -18.508, 90.01, 0, 18.497, 74.905]
  MoveL 8891 to (-70.21, 28.6, -14.75) mm, rotated rx 180 ry 0 rz 90 deg; joints [74.093, -18.411, 89.567, 0, 18.844, 74.093]
  MoveL 8892 to (-62.66, 28.6, -14.75) mm, rotated rx -180 ry 0 rz 90 deg; joints [74.166, -18.299, 89.06, 0, 19.239, 74.166]
  MoveL 8893 to (-62.66, 28.6, -11.75) mm, rotated rx -180 ry 0 rz 90 deg; joints [74.166, -18.456, 89.163, 0, 19.293, 74.166]
  Establecer velocidad (1000.0 mm/s)
  MoveL 8894 to (-62.66, 28.6, 10) mm, rotated rx -180 ry 0 rz 90 deg; joints [74.166, -19.592, 89.893, 0, 19.699, 74.166]
  Establecer velocidad (66.7 mm/s)
  MoveL 8895 to (2.53, 61.18, 10) mm, rotated rx 180 ry 0 rz 90 deg; joints [75.833, -18.643, 85.994, 0, 22.649, 75.833]
  MoveL 8896 to (2.53, 61.18, -11.5) mm, rotated rx -180 ry 0 rz 90 deg; joints [75.833, -17.539, 85.273, 0, 22.266, 75.833]
  MoveL 8897 to (2.53, 68.09, -13.35) mm, rotated rx 180 ry 0 rz 90 deg; joints [76.061, -17.475, 85.332, 0, 22.143, 76.061]
  MoveL 8898 to (0.47, 68.19, -13.9) mm, rotated rx -180 ry 0 rz 90 deg; joints [76.047, -17.483, 85.46, 0, 22.023, 76.047]
  MoveL 8899 to (-2.68, 68.32, -14.75) mm, rotated rx 180 ry 0 rz 90 deg; joints [76.026, -17.495, 85.656, 0, 21.84, 76.026]
  MoveL 8900 to (-7.89, 68.53, -14.75) mm, rotated rx -180 ry 0 rz 90 deg; joints [75.99, -17.587, 86.026, 0, 21.561, 75.99]
  MoveC 8901 to (-9.75, 66.22, -14.75) mm, rotated rx 180 ry 0 rz 90 deg; joints [75.898, -17.609, 86.115, 0, 21.493, 75.898] to (-9.56, 63.27, -14.75) mm, rotated rx 180 ry 0 rz 90 deg; joints [75.801, -17.593, 86.05, 0, 21.543, 75.801]
  MoveC 8902 to (-6.43, 61.14, -14.75) mm, rotated rx -180 ry 0 rz 90 deg; joints [75.757, -17.529, 85.792, 0, 21.737, 75.757] to (-3.32, 58.97, -14.75) mm, rotated rx -180 ry 0 rz 90 deg; joints [75.712, -17.465, 85.535, 0, 21.931, 75.712]
  MoveL 8903 to (-2.5, 58.94, -14.75) mm, rotated rx -180 ry 0 rz 90 deg; joints [75.718, -17.451, 85.477, 0, 21.974, 75.718]
  MoveL 8904 to (-2.37, 58.96, -14.75) mm, rotated rx -180 ry 0 rz 90 deg; joints [75.719, -17.449, 85.468, 0, 21.981, 75.719]
  MoveC 8905 to (0.08, 59.21, -14.75) mm, rotated rx 180 ry 0 rz 90 deg; joints [75.748, -17.406, 85.299, 0, 22.107, 75.748] to (2.53, 59.51, -14.75) mm, rotated rx 180 ry 0 rz 90 deg; joints [75.778, -17.364, 85.131, 0, 22.233, 75.778]
  MoveL 8906 to (2.53, 68.09, -14.75) mm, rotated rx 180 ry 0 rz 90 deg; joints [76.061, -17.403, 85.284, 0, 22.119, 76.061]
  MoveL 8907 to (0.47, 68.19, -14.75) mm, rotated rx 180 ry 0 rz 90 deg; joints [76.047, -17.439, 85.431, 0, 22.009, 76.047]
  MoveL 8908 to (-2.68, 68.32, -14.75) mm, rotated rx 180 ry 0 rz 90 deg; joints [76.026, -17.495, 85.656, 0, 21.84, 76.026]
  MoveL 8909 to (-2.99, 60.78, -14.75) mm, rotated rx -180 ry 0 rz 90 deg; joints [75.774, -17.467, 85.544, 0, 21.924, 75.774]
  MoveL 8910 to (-2.99, 60.78, -11.75) mm, rotated rx 180 ry 0 rz 90 deg; joints [75.774, -17.622, 85.646, 0, 21.976, 75.774]
  Establecer velocidad (1000.0 mm/s)
  MoveL 8911 to (-2.99, 60.78, 10) mm, rotated rx 180 ry 0 rz 90 deg; joints [75.774, -18.74, 86.376, 0, 22.364, 75.774]
  Establecer velocidad (66.7 mm/s)
  MoveL 8912 to (-3.8, 68.19, 10) mm, rotated rx -180 ry 0 rz 90 deg; joints [76.012, -18.788, 86.565, 0, 22.223, 76.012]
  MoveL 8913 to (-3.8, 68.19, -11.75) mm, rotated rx -180 ry 0 rz 90 deg; joints [76.012, -17.669, 85.835, 0, 21.834, 76.012]
  MoveL 8914 to (-3.8, 68.19, -15) mm, rotated rx 180 ry 0 rz 90 deg; joints [76.012, -17.501, 85.724, 0, 21.778, 76.012]
  MoveL 8915 to (-7.27, 68.33, -15) mm, rotated rx -180 ry 0 rz 90 deg; joints [75.988, -17.562, 85.97, 0, 21.592, 75.988]
  MoveC 8916 to (-9.1, 66.05, -15) mm, rotated rx -180 ry 0 rz 90 deg; joints [75.897, -17.584, 86.058, 0, 21.525, 75.897] to (-8.92, 63.13, -15) mm, rotated rx 180 ry 0 rz 90 deg; joints [75.802, -17.568, 85.994, 0, 21.574, 75.802]
  MoveL 8917 to (-4.6, 60.18, -15) mm, rotated rx 180 ry 0 rz 90 deg; joints [75.741, -17.48, 85.638, 0, 21.842, 75.741]
  MoveL 8918 to (-3.29, 59.21, -15) mm, rotated rx 180 ry 0 rz 90 deg; joints [75.72, -17.453, 85.528, 0, 21.925, 75.72]
  MoveC 8919 to (-3.11, 59.1, -15) mm, rotated rx 180 ry 0 rz 90 deg; joints [75.718, -17.449, 85.514, 0, 21.935, 75.718] to (-2.92, 59.03, -15) mm, rotated rx 180 ry 0 rz 90 deg; joints [75.717, -17.446, 85.499, 0, 21.947, 75.717]
  MoveL 8920 to (-2.85, 59.02, -15) mm, rotated rx -180 ry 0 rz 90 deg; joints [75.717, -17.444, 85.494, 0, 21.95, 75.717]
  MoveL 8921 to (-0.33, 59.28, -15) mm, rotated rx 180 ry 0 rz 90 deg; joints [75.747, -17.401, 85.321, 0, 22.08, 75.747]
  MoveL 8922 to (-0.33, 68.05, -15) mm, rotated rx -180 ry 0 rz 90 deg; joints [76.036, -17.44, 85.476, 0, 21.964, 76.036]
  MoveL 8923 to (-3.8, 68.19, -15) mm, rotated rx 180 ry 0 rz 90 deg; joints [76.012, -17.501, 85.724, 0, 21.778, 76.012]
  MoveL 8924 to (-4.11, 60.65, -15) mm, rotated rx -180 ry 0 rz 90 deg; joints [75.76, -17.474, 85.612, 0, 21.862, 75.76]
  MoveL 8925 to (-4.11, 60.65, -12) mm, rotated rx -180 ry 0 rz 90 deg; joints [75.76, -17.628, 85.714, 0, 21.914, 75.76]
  Establecer velocidad (1000.0 mm/s)
  MoveL 8926 to (-4.11, 60.65, 10) mm, rotated rx 180 ry 0 rz 90 deg; joints [75.76, -18.76, 86.453, 0, 22.307, 75.76]
  Establecer velocidad (66.7 mm/s)
  MoveL 8927 to (-61.8, 35.68, 10) mm, rotated rx -180 ry 0 rz 90 deg; joints [74.413, -19.61, 89.97, 0, 19.64, 74.413]
  MoveL 8928 to (-61.8, 35.68, -11.75) mm, rotated rx -180 ry 0 rz 90 deg; joints [74.413, -18.473, 89.239, 0, 19.233, 74.413]
  MoveL 8929 to (-63.31, 35.86, -12.16) mm, rotated rx 180 ry 0 rz 90 deg; joints [74.405, -18.475, 89.331, 0, 19.145, 74.405]
  MoveL 8930 to (-64.82, 35.68, -12.56) mm, rotated rx -180 ry 0 rz 90 deg; joints [74.385, -18.476, 89.415, 0, 19.061, 74.385]
  MoveL 8931 to (-66.25, 35.17, -12.97) mm, rotated rx 180 ry 0 rz 90 deg; joints [74.354, -18.473, 89.487, 0, 18.986, 74.354]
  MoveL 8932 to (-67.53, 34.35, -13.38) mm, rotated rx -180 ry 0 rz 90 deg; joints [74.314, -18.468, 89.544, 0, 18.924, 74.314]
  MoveL 8933 to (-68.6, 33.27, -13.78) mm, rotated rx -180 ry 0 rz 90 deg; joints [74.267, -18.458, 89.581, 0, 18.876, 74.267]
  MoveL 8934 to (-69.41, 31.98, -14.19) mm, rotated rx -180 ry 0 rz 90 deg; joints [74.216, -18.443, 89.597, 0, 18.846, 74.216]
  MoveL 8935 to (-69.9, 30.55, -14.59) mm, rotated rx -180 ry 0 rz 90 deg; joints [74.162, -18.423, 89.589, 0, 18.834, 74.162]
  MoveL 8936 to (-70.04, 29.04, -15) mm, rotated rx 180 ry 0 rz 90 deg; joints [74.11, -18.397, 89.556, 0, 18.841, 74.11]
  MoveL 8937 to (-70.04, 5.21, -15) mm, rotated rx 180 ry 0 rz 90 deg; joints [73.306, -18.294, 89.089, 0, 19.205, 73.306]
  MoveC 8938 to (-69.06, 3.13, -15) mm, rotated rx -180 ry 0 rz 90 deg; joints [73.246, -18.27, 88.981, 0, 19.289, 73.246] to (-66.81, 2.63, -15) mm, rotated rx 180 ry 0 rz 90 deg; joints [73.252, -18.234, 88.82, 0, 19.414, 73.252]
  MoveC 8939 to (-46.89, 7.49, -15) mm, rotated rx -180 ry 0 rz 90 deg; joints [73.612, -17.946, 87.569, 0, 20.377, 73.612] to (-27.01, 12.48, -15) mm, rotated rx 180 ry 0 rz 90 deg; joints [73.968, -17.643, 86.301, 0, 21.342, 73.968]
  MoveL 8940 to (-26.06, 12.75, -15) mm, rotated rx 180 ry 0 rz 90 deg; joints [73.986, -17.628, 86.241, 0, 21.387, 73.986]
  MoveC 8941 to (-24.7, 14.16, -15) mm, rotated rx -180 ry 0 rz 90 deg; joints [74.045, -17.612, 86.175, 0, 21.437, 74.045] to (-24.5, 16.11, -15) mm, rotated rx -180 ry 0 rz 90 deg; joints [74.111, -17.618, 86.2, 0, 21.419, 74.111]
  MoveL 8942 to (-24.65, 16.58, -15) mm, rotated rx 180 ry 0 rz 90 deg; joints [74.125, -17.623, 86.219, 0, 21.404, 74.125]
  MoveL 8943 to (-29.09, 29.24, -15) mm, rotated rx -180 ry 0 rz 90 deg; joints [74.502, -17.757, 86.773, 0, 20.984, 74.502]
  MoveC 8944 to (-29.52, 30.04, -15) mm, rotated rx 180 ry 0 rz 90 deg; joints [74.525, -17.768, 86.818, 0, 20.95, 74.525] to (-30.2, 30.67, -15) mm, rotated rx 180 ry 0 rz 90 deg; joints [74.539, -17.782, 86.877, 0, 20.905, 74.539]
  MoveC 8945 to (-48.18, 42.62, -15) mm, rotated rx -180 ry 0 rz 90 deg; joints [74.774, -18.124, 88.335, 0, 19.789, 74.774] to (-66.23, 54.49, -15) mm, rotated rx -180 ry 0 rz 90 deg; joints [75.011, -18.445, 89.772, 0, 18.673, 75.011]
  MoveC 8946 to (-68.39, 54.35, -15) mm, rotated rx 180 ry 0 rz 90 deg; joints [74.986, -18.476, 89.914, 0, 18.562, 74.986] to (-69.95, 52.85, -15) mm, rotated rx 180 ry 0 rz 90 deg; joints [74.921, -18.492, 89.992, 0, 18.501, 74.921]
  MoveL 8947 to (-70.04, 52.42, -15) mm, rotated rx -180 ry 0 rz 90 deg; joints [74.905, -18.492, 89.99, 0, 18.502, 74.905]
  MoveL 8948 to (-70.04, 51.65, -15) mm, rotated rx -180 ry 0 rz 90 deg; joints [74.879, -18.489, 89.976, 0, 18.513, 74.879]
  MoveL 8949 to (-70.04, 29.04, -15) mm, rotated rx 180 ry 0 rz 90 deg; joints [74.11, -18.397, 89.556, 0, 18.841, 74.11]
  MoveL 8950 to (-62.49, 29.04, -15) mm, rotated rx 180 ry 0 rz 90 deg; joints [74.182, -18.285, 89.049, 0, 19.236, 74.182]
  MoveL 8951 to (-62.49, 29.04, -12) mm, rotated rx -180 ry 0 rz 90 deg; joints [74.182, -18.442, 89.152, 0, 19.291, 74.182]
  Establecer velocidad (1000.0 mm/s)
  MoveL 8952 to (-62.49, 29.04, 10) mm, rotated rx 180 ry 0 rz 90 deg; joints [74.182, -19.591, 89.89, 0, 19.701, 74.182]
  Establecer velocidad (66.7 mm/s)
  MoveL 8953 to (-40.21, -35.65, 10) mm, rotated rx -180 ry 0 rz 90 deg; joints [72.26, -18.909, 87.045, 0, 21.864, 72.26]
  MoveL 8954 to (-40.21, -35.65, -11.75) mm, rotated rx -180 ry 0 rz 90 deg; joints [72.26, -17.787, 86.315, 0, 21.472, 72.26]
  MoveL 8955 to (-40.31, -34.13, -12.16) mm, rotated rx -180 ry 0 rz 90 deg; joints [72.308, -17.776, 86.342, 0, 21.434, 72.308]
  MoveL 8956 to (-40.78, -32.69, -12.56) mm, rotated rx 180 ry 0 rz 90 deg; joints [72.35, -17.771, 86.392, 0, 21.379, 72.35]
  MoveL 8957 to (-41.56, -31.38, -12.97) mm, rotated rx -180 ry 0 rz 90 deg; joints [72.385, -17.77, 86.46, 0, 21.31, 72.385]
  MoveL 8958 to (-42.6, -30.28, -13.38) mm, rotated rx -180 ry 0 rz 90 deg; joints [72.41, -17.772, 86.542, 0, 21.23, 72.41]
  MoveL 8959 to (-43.87, -29.44, -13.78) mm, rotated rx -180 ry 0 rz 90 deg; joints [72.424, -17.776, 86.633, 0, 21.144, 72.424]
  MoveL 8960 to (-45.29, -28.9, -14.19) mm, rotated rx 180 ry 0 rz 90 deg; joints [72.427, -17.782, 86.728, 0, 21.054, 72.427]
  MoveL 8961 to (-46.79, -28.68, -14.59) mm, rotated rx 180 ry 0 rz 90 deg; joints [72.419, -17.787, 86.822, 0, 20.965, 72.419]
  MoveL 8962 to (-48.3, -28.83, -15) mm, rotated rx 180 ry 0 rz 90 deg; joints [72.398, -17.789, 86.907, 0, 20.882, 72.398]
  MoveC 8963 to (-58.16, -30.77, -15) mm, rotated rx -180 ry 0 rz 90 deg; joints [72.231, -17.938, 87.536, 0, 20.402, 72.231] to (-68.01, -32.74, -15) mm, rotated rx -180 ry 0 rz 90 deg; joints [72.061, -18.083, 88.158, 0, 19.925, 72.061]
  MoveC 8964 to (-69.45, -33.59, -15) mm, rotated rx 180 ry 0 rz 90 deg; joints [72.018, -18.101, 88.236, 0, 19.865, 72.018] to (-70.04, -35.16, -15) mm, rotated rx -180 ry 0 rz 90 deg; joints [71.959, -18.102, 88.242, 0, 19.861, 71.959]
  MoveL 8965 to (-70.04, -35.54, -15) mm, rotated rx 180 ry 0 rz 90 deg; joints [71.947, -18.1, 88.234, 0, 19.867, 71.947]
  MoveL 8966 to (-70.04, -67.21, -15) mm, rotated rx 180 ry 0 rz 90 deg; joints [70.905, -17.934, 87.518, 0, 20.416, 70.905]
  MoveC 8967 to (-70.02, -67.58, -15) mm, rotated rx -180 ry 0 rz 90 deg; joints [70.893, -17.932, 87.508, 0, 20.424, 70.893] to (-69.96, -67.95, -15) mm, rotated rx 180 ry 0 rz 90 deg; joints [70.881, -17.929, 87.495, 0, 20.433, 70.881]
  MoveC 8968 to (-69.09, -69.32, -15) mm, rotated rx 180 ry 0 rz 90 deg; joints [70.846, -17.908, 87.405, 0, 20.503, 70.846] to (-67.55, -69.87, -15) mm, rotated rx 180 ry 0 rz 90 deg; joints [70.846, -17.88, 87.289, 0, 20.591, 70.846]
  MoveL 8969 to (-66.81, -69.88, -15) mm, rotated rx 180 ry 0 rz 90 deg; joints [70.854, -17.868, 87.238, 0, 20.63, 70.854]
  MoveL 8970 to (-61.12, -69.75, -15) mm, rotated rx -180 ry 0 rz 90 deg; joints [70.922, -17.777, 86.857, 0, 20.92, 70.922]
  MoveL 8971 to (-60.18, -69.74, -15) mm, rotated rx 180 ry 0 rz 90 deg; joints [70.934, -17.762, 86.793, 0, 20.969, 70.934]
  MoveL 8972 to (-39.33, -69.24, -15) mm, rotated rx -180 ry 0 rz 90 deg; joints [71.181, -17.416, 85.38, 0, 22.036, 71.181]
  MoveL 8973 to (-37.91, -69.18, -15) mm, rotated rx -180 ry 0 rz 90 deg; joints [71.198, -17.392, 85.283, 0, 22.109, 71.198]
  MoveC 8974 to (-36.44, -68.65, -15) mm, rotated rx 180 ry 0 rz 90 deg; joints [71.232, -17.369, 85.194, 0, 22.175, 71.232] to (-35.54, -67.37, -15) mm, rotated rx -180 ry 0 rz 90 deg; joints [71.282, -17.361, 85.162, 0, 22.2, 71.282]
  MoveL 8975 to (-35.36, -66.81, -15) mm, rotated rx 180 ry 0 rz 90 deg; joints [71.302, -17.362, 85.163, 0, 22.199, 71.302]
  MoveL 8976 to (-34.59, -63.76, -15) mm, rotated rx 180 ry 0 rz 90 deg; joints [71.409, -17.366, 85.18, 0, 22.186, 71.409]
  MoveL 8977 to (-25.58, -28.43, -15) mm, rotated rx -180 ry 0 rz 90 deg; joints [72.645, -17.409, 85.35, 0, 22.058, 72.645]
  MoveL 8978 to (-25.54, -28.24, -15) mm, rotated rx -180 ry 0 rz 90 deg; joints [72.651, -17.409, 85.352, 0, 22.057, 72.651]
  MoveC 8979 to (-26.29, -26.34, -15) mm, rotated rx 180 ry 0 rz 90 deg; joints [72.706, -17.432, 85.445, 0, 21.987, 72.706] to (-27.92, -25.1, -15) mm, rotated rx 180 ry 0 rz 90 deg; joints [72.729, -17.467, 85.585, 0, 21.882, 72.729]
  MoveC 8980 to (-28.24, -25.02, -15) mm, rotated rx -180 ry 0 rz 90 deg; joints [72.729, -17.473, 85.609, 0, 21.864, 72.729] to (-28.57, -25.03, -15) mm, rotated rx -180 ry 0 rz 90 deg; joints [72.725, -17.479, 85.632, 0, 21.847, 72.725]
  MoveC 8981 to (-38.44, -26.92, -15) mm, rotated rx -180 ry 0 rz 90 deg; joints [72.563, -17.636, 86.273, 0, 21.363, 72.563] to (-48.3, -28.83, -15) mm, rotated rx 180 ry 0 rz 90 deg; joints [72.398, -17.789, 86.907, 0, 20.882, 72.398]
  MoveL 8982 to (-46.86, -36.24, -15) mm, rotated rx 180 ry 0 rz 90 deg; joints [72.171, -17.727, 86.647, 0, 21.08, 72.171]
  MoveL 8983 to (-46.86, -36.24, -12) mm, rotated rx -180 ry 0 rz 90 deg; joints [72.171, -17.882, 86.75, 0, 21.133, 72.171]
  Establecer velocidad (1000.0 mm/s)
  MoveL 8984 to (-46.86, -36.24, 10) mm, rotated rx -180 ry 0 rz 90 deg; joints [72.171, -19.019, 87.488, 0, 21.531, 72.171]
  Establecer velocidad (66.7 mm/s)
  MoveL 8985 to (-40.16, -35.79, 10) mm, rotated rx 180 ry 0 rz 90 deg; joints [72.255, -18.907, 87.039, 0, 21.869, 72.255]
  MoveL 8986 to (-40.16, -35.79, -12) mm, rotated rx 180 ry 0 rz 90 deg; joints [72.255, -17.773, 86.301, 0, 21.472, 72.255]
  MoveL 8987 to (-40.27, -34.28, -12.41) mm, rotated rx -180 ry 0 rz 90 deg; joints [72.303, -17.762, 86.327, 0, 21.434, 72.303]
  MoveL 8988 to (-40.74, -32.84, -12.81) mm, rotated rx 180 ry 0 rz 90 deg; joints [72.346, -17.757, 86.377, 0, 21.379, 72.346]
  MoveL 8989 to (-41.52, -31.53, -13.22) mm, rotated rx -180 ry 0 rz 90 deg; joints [72.38, -17.756, 86.446, 0, 21.31, 72.38]
  MoveL 8990 to (-42.57, -30.43, -13.62) mm, rotated rx 180 ry 0 rz 90 deg; joints [72.405, -17.758, 86.528, 0, 21.23, 72.405]
  MoveL 8991 to (-43.84, -29.59, -14.03) mm, rotated rx -180 ry 0 rz 90 deg; joints [72.42, -17.762, 86.619, 0, 21.143, 72.42]
  MoveL 8992 to (-45.26, -29.05, -14.44) mm, rotated rx -180 ry 0 rz 90 deg; joints [72.423, -17.767, 86.714, 0, 21.054, 72.423]
  MoveL 8993 to (-46.76, -28.84, -14.84) mm, rotated rx 180 ry 0 rz 90 deg; joints [72.414, -17.772, 86.808, 0, 20.965, 72.414]
  MoveL 8994 to (-48.27, -28.99, -15.25) mm, rotated rx -180 ry 0 rz 90 deg; joints [72.393, -17.775, 86.893, 0, 20.882, 72.393]
  MoveL 8995 to (-65.86, -32.46, -15.25) mm, rotated rx -180 ry 0 rz 90 deg; joints [72.093, -18.038, 88.011, 0, 20.027, 72.093]
  MoveL 8996 to (-67.87, -32.86, -15.25) mm, rotated rx 180 ry 0 rz 90 deg; joints [72.059, -18.067, 88.138, 0, 19.93, 72.059]
  MoveC 8997 to (-69.31, -33.73, -15.25) mm, rotated rx 180 ry 0 rz 90 deg; joints [72.014, -18.085, 88.216, 0, 19.87, 72.014] to (-69.88, -35.32, -15.25) mm, rotated rx -180 ry 0 rz 90 deg; joints [71.956, -18.086, 88.219, 0, 19.867, 71.956]
  MoveL 8998 to (-69.88, -67.18, -15.25) mm, rotated rx -180 ry 0 rz 90 deg; joints [70.907, -17.919, 87.499, 0, 20.419, 70.907]
  MoveC 8999 to (-69.83, -67.71, -15.25) mm, rotated rx 180 ry 0 rz 90 deg; joints [70.891, -17.915, 87.484, 0, 20.432, 70.891] to (-69.67, -68.23, -15.25) mm, rotated rx 180 ry 0 rz 90 deg; joints [70.875, -17.91, 87.461, 0, 20.449, 70.875]
  MoveC 9000 to (-68.77, -69.29, -15.25) mm, rotated rx -180 ry 0 rz 90 deg; joints [70.851, -17.89, 87.376, 0, 20.514, 70.851] to (-67.44, -69.72, -15.25) mm, rotated rx 180 ry 0 rz 90 deg; joints [70.852, -17.866, 87.276, 0, 20.59, 70.852]
  MoveC 9001 to (-67.04, -69.73, -15.25) mm, rotated rx -180 ry 0 rz 90 deg; joints [70.856, -17.86, 87.249, 0, 20.611, 70.856] to (-66.64, -69.73, -15.25) mm, rotated rx 180 ry 0 rz 90 deg; joints [70.861, -17.853, 87.222, 0, 20.631, 70.861]
  MoveC 9002 to (-52.36, -69.41, -15.25) mm, rotated rx 180 ry 0 rz 90 deg; joints [71.031, -17.622, 86.261, 0, 21.362, 71.031] to (-38.08, -69.03, -15.25) mm, rotated rx 180 ry 0 rz 90 deg; joints [71.201, -17.383, 85.29, 0, 22.093, 71.201]
  MoveC 9003 to (-36.49, -68.45, -15.25) mm, rotated rx 180 ry 0 rz 90 deg; joints [71.237, -17.359, 85.194, 0, 22.165, 71.237] to (-35.57, -67.02, -15.25) mm, rotated rx -180 ry 0 rz 90 deg; joints [71.293, -17.351, 85.163, 0, 22.188, 71.293]
  MoveL 9004 to (-25.86, -28.9, -15.25) mm, rotated rx 180 ry 0 rz 90 deg; joints [72.627, -17.398, 85.351, 0, 22.047, 72.627]
  MoveC 9005 to (-25.79, -28.18, -15.25) mm, rotated rx 180 ry 0 rz 90 deg; joints [72.651, -17.401, 85.362, 0, 22.039, 72.651] to (-25.96, -27.48, -15.25) mm, rotated rx -180 ry 0 rz 90 deg; joints [72.672, -17.407, 85.389, 0, 22.019, 72.672]
  MoveL 9006 to (-26.06, -27.25, -15.25) mm, rotated rx -180 ry 0 rz 90 deg; joints [72.678, -17.41, 85.401, 0, 22.01, 72.678]
  MoveC 9007 to (-27.04, -25.95, -15.25) mm, rotated rx 180 ry 0 rz 90 deg; joints [72.711, -17.435, 85.498, 0, 21.937, 72.711] to (-28.51, -25.22, -15.25) mm, rotated rx -180 ry 0 rz 90 deg; joints [72.719, -17.464, 85.615, 0, 21.849, 72.719]
  MoveL 9008 to (-29.85, -25.45, -15.25) mm, rotated rx -180 ry 0 rz 90 deg; joints [72.698, -17.485, 85.703, 0, 21.783, 72.698]
  MoveL 9009 to (-46.91, -28.72, -15.25) mm, rotated rx -180 ry 0 rz 90 deg; joints [72.416, -17.754, 86.806, 0, 20.948, 72.416]
  MoveL 9010 to (-48.27, -28.99, -15.25) mm, rotated rx -180 ry 0 rz 90 deg; joints [72.393, -17.775, 86.893, 0, 20.882, 72.393]
  MoveL 9011 to (-46.81, -36.4, -15.25) mm, rotated rx -180 ry 0 rz 90 deg; joints [72.166, -17.712, 86.632, 0, 21.081, 72.166]
  MoveL 9012 to (-46.81, -36.4, -12.25) mm, rotated rx -180 ry 0 rz 90 deg; joints [72.166, -17.868, 86.734, 0, 21.133, 72.166]
  Establecer velocidad (1000.0 mm/s)
  MoveL 9013 to (-46.81, -36.4, 10) mm, rotated rx -180 ry 0 rz 90 deg; joints [72.166, -19.017, 87.481, 0, 21.536, 72.166]
  Establecer velocidad (66.7 mm/s)
  MoveL 9014 to (-61.64, 35.34, 10) mm, rotated rx -180 ry 0 rz 90 deg; joints [74.403, -19.606, 89.952, 0, 19.653, 74.403]
  MoveL 9015 to (-61.64, 35.34, -12) mm, rotated rx -180 ry 0 rz 90 deg; joints [74.403, -18.456, 89.213, 0, 19.242, 74.403]
  MoveL 9016 to (-63.14, 35.52, -12.41) mm, rotated rx 180 ry 0 rz 90 deg; joints [74.395, -18.458, 89.305, 0, 19.154, 74.395]
  MoveL 9017 to (-64.65, 35.34, -12.81) mm, rotated rx 180 ry 0 rz 90 deg; joints [74.375, -18.459, 89.389, 0, 19.07, 74.375]
  MoveL 9018 to (-66.08, 34.83, -13.22) mm, rotated rx 180 ry 0 rz 90 deg; joints [74.344, -18.457, 89.461, 0, 18.995, 74.344]
  MoveL 9019 to (-67.37, 34.01, -13.62) mm, rotated rx -180 ry 0 rz 90 deg; joints [74.304, -18.451, 89.518, 0, 18.933, 74.304]
  MoveL 9020 to (-68.44, 32.93, -14.03) mm, rotated rx 180 ry 0 rz 90 deg; joints [74.257, -18.441, 89.556, 0, 18.885, 74.257]
  MoveL 9021 to (-69.24, 31.65, -14.44) mm, rotated rx -180 ry 0 rz 90 deg; joints [74.206, -18.426, 89.571, 0, 18.855, 74.206]
  MoveL 9022 to (-69.74, 30.21, -14.84) mm, rotated rx -180 ry 0 rz 90 deg; joints [74.152, -18.406, 89.563, 0, 18.843, 74.152]
  MoveL 9023 to (-69.88, 28.7, -15.25) mm, rotated rx -180 ry 0 rz 90 deg; joints [74.1, -18.381, 89.53, 0, 18.851, 74.1]
  MoveL 9024 to (-69.88, 6.16, -15.25) mm, rotated rx -180 ry 0 rz 90 deg; joints [73.339, -18.283, 89.089, 0, 19.194, 73.339]
  MoveL 9025 to (-69.88, 5.21, -15.25) mm, rotated rx -180 ry 0 rz 90 deg; joints [73.308, -18.279, 89.07, 0, 19.209, 73.308]
  MoveC 9026 to (-68.83, 3.25, -15.25) mm, rotated rx -180 ry 0 rz 90 deg; joints [73.252, -18.254, 88.96, 0, 19.294, 73.252] to (-66.66, 2.8, -15.25) mm, rotated rx 180 ry 0 rz 90 deg; joints [73.259, -18.219, 88.805, 0, 19.414, 73.259]
  MoveC 9027 to (-46.71, 7.69, -15.25) mm, rotated rx 180 ry 0 rz 90 deg; joints [73.62, -17.931, 87.552, 0, 20.379, 73.62] to (-26.79, 12.71, -15.25) mm, rotated rx 180 ry 0 rz 90 deg; joints [73.977, -17.628, 86.282, 0, 21.346, 73.977]
  MoveC 9028 to (-24.96, 14.14, -15.25) mm, rotated rx 180 ry 0 rz 90 deg; joints [74.042, -17.604, 86.184, 0, 21.42, 74.042] to (-24.78, 16.46, -15.25) mm, rotated rx -180 ry 0 rz 90 deg; joints [74.12, -17.612, 86.217, 0, 21.395, 74.12]
  MoveL 9029 to (-29.21, 29.12, -15.25) mm, rotated rx 180 ry 0 rz 90 deg; joints [74.497, -17.746, 86.77, 0, 20.975, 74.497]
  MoveC 9030 to (-29.65, 29.93, -15.25) mm, rotated rx -180 ry 0 rz 90 deg; joints [74.52, -17.757, 86.816, 0, 20.94, 74.52] to (-30.33, 30.56, -15.25) mm, rotated rx -180 ry 0 rz 90 deg; joints [74.535, -17.771, 86.875, 0, 20.896, 74.535]
  MoveC 9031 to (-48.06, 42.37, -15.25) mm, rotated rx 180 ry 0 rz 90 deg; joints [74.766, -18.108, 88.314, 0, 19.794, 74.766] to (-65.86, 54.09, -15.25) mm, rotated rx 180 ry 0 rz 90 deg; joints [75, -18.425, 89.731, 0, 18.693, 75]
  MoveC 9032 to (-66.31, 54.32, -15.25) mm, rotated rx -180 ry 0 rz 90 deg; joints [75.004, -18.432, 89.766, 0, 18.667, 75.004] to (-66.81, 54.39, -15.25) mm, rotated rx 180 ry 0 rz 90 deg; joints [75.002, -18.44, 89.8, 0, 18.639, 75.002]
  MoveC 9033 to (-68.08, 54.16, -15.25) mm, rotated rx -180 ry 0 rz 90 deg; joints [74.982, -18.457, 89.881, 0, 18.576, 74.982] to (-69.18, 53.48, -15.25) mm, rotated rx -180 ry 0 rz 90 deg; joints [74.949, -18.471, 89.943, 0, 18.528, 74.949]
  MoveL 9034 to (-69.64, 52.89, -15.25) mm, rotated rx -180 ry 0 rz 90 deg; joints [74.925, -18.475, 89.963, 0, 18.512, 74.925]
  MoveC 9035 to (-69.82, 52.56, -15.25) mm, rotated rx -180 ry 0 rz 90 deg; joints [74.912, -18.476, 89.969, 0, 18.507, 74.912] to (-69.88, 52.19, -15.25) mm, rotated rx 180 ry 0 rz 90 deg; joints [74.898, -18.476, 89.966, 0, 18.509, 74.898]
  MoveL 9036 to (-69.88, 28.7, -15.25) mm, rotated rx -180 ry 0 rz 90 deg; joints [74.1, -18.381, 89.53, 0, 18.851, 74.1]
  MoveL 9037 to (-62.33, 28.7, -15.25) mm, rotated rx 180 ry 0 rz 90 deg; joints [74.172, -18.268, 89.023, 0, 19.245, 74.172]
  MoveL 9038 to (-62.33, 28.7, -12.25) mm, rotated rx -180 ry 0 rz 90 deg; joints [74.172, -18.425, 89.126, 0, 19.299, 74.172]
  Establecer velocidad (1000.0 mm/s)
  MoveL 9039 to (-62.33, 28.7, 10) mm, rotated rx -180 ry 0 rz 90 deg; joints [74.172, -19.587, 89.873, 0, 19.714, 74.172]
  Establecer velocidad (66.7 mm/s)
  MoveL 9040 to (-3.19, 63.69, 10) mm, rotated rx -180 ry 0 rz 90 deg; joints [75.869, -18.757, 86.442, 0, 22.315, 75.869]
  MoveL 9041 to (-3.19, 63.69, -12) mm, rotated rx 180 ry 0 rz 90 deg; joints [75.869, -17.626, 85.704, 0, 21.922, 75.869]
  MoveL 9042 to (-3.19, 63.69, -15.25) mm, rotated rx 180 ry 0 rz 90 deg; joints [75.869, -17.458, 85.592, 0, 21.866, 75.869]
  MoveL 9043 to (-3.19, 67.98, -15.25) mm, rotated rx 180 ry 0 rz 90 deg; joints [76.01, -17.477, 85.668, 0, 21.809, 76.01]
  MoveL 9044 to (-6.68, 68.13, -15.25) mm, rotated rx 180 ry 0 rz 90 deg; joints [75.986, -17.538, 85.917, 0, 21.622, 75.986]
  MoveC 9045 to (-8.46, 65.87, -15.25) mm, rotated rx 180 ry 0 rz 90 deg; joints [75.897, -17.559, 86.002, 0, 21.557, 75.897] to (-8.28, 63, -15.25) mm, rotated rx 180 ry 0 rz 90 deg; joints [75.803, -17.544, 85.939, 0, 21.605, 75.803]
  MoveC 9046 to (-5.71, 61.24, -15.25) mm, rotated rx 180 ry 0 rz 90 deg; joints [75.766, -17.491, 85.726, 0, 21.765, 75.766] to (-3.19, 59.4, -15.25) mm, rotated rx -180 ry 0 rz 90 deg; joints [75.727, -17.439, 85.516, 0, 21.923, 75.727]
  MoveL 9047 to (-3.19, 63.69, -15.25) mm, rotated rx 180 ry 0 rz 90 deg; joints [75.869, -17.458, 85.592, 0, 21.866, 75.869]
  MoveL 9048 to (-6.96, 63.69, -15.25) mm, rotated rx -180 ry 0 rz 90 deg; joints [75.837, -17.524, 85.858, 0, 21.666, 75.837]
  MoveL 9049 to (-6.96, 63.69, -12.25) mm, rotated rx 180 ry 0 rz 90 deg; joints [75.837, -17.679, 85.961, 0, 21.718, 75.837]
  Establecer velocidad (1000.0 mm/s)
  MoveL 9050 to (-6.96, 63.69, 10) mm, rotated rx -180 ry 0 rz 90 deg; joints [75.837, -18.824, 86.708, 0, 22.117, 75.837]
  Establecer velocidad (66.7 mm/s)
  MoveL 9051 to (-6.05, 64.85, 10) mm, rotated rx 180 ry 0 rz 90 deg; joints [75.883, -18.813, 86.664, 0, 22.15, 75.883]
  MoveL 9052 to (-6.05, 64.85, -12.25) mm, rotated rx -180 ry 0 rz 90 deg; joints [75.883, -17.668, 85.917, 0, 21.751, 75.883]
  MoveL 9053 to (-6.05, 64.85, -15.5) mm, rotated rx 180 ry 0 rz 90 deg; joints [75.883, -17.5, 85.806, 0, 21.695, 75.883]
  MoveL 9054 to (-6.05, 67.93, -15.5) mm, rotated rx 180 ry 0 rz 90 deg; joints [75.985, -17.514, 85.86, 0, 21.654, 75.985]
  MoveC 9055 to (-7.81, 65.7, -15.5) mm, rotated rx 180 ry 0 rz 90 deg; joints [75.897, -17.534, 85.945, 0, 21.589, 75.897] to (-7.64, 62.86, -15.5) mm, rotated rx -180 ry 0 rz 90 deg; joints [75.804, -17.519, 85.882, 0, 21.637, 75.804]
  MoveL 9056 to (-6.05, 61.76, -15.5) mm, rotated rx 180 ry 0 rz 90 deg; joints [75.781, -17.487, 85.751, 0, 21.736, 75.781]
  MoveL 9057 to (-6.05, 64.85, -15.5) mm, rotated rx 180 ry 0 rz 90 deg; joints [75.883, -17.5, 85.806, 0, 21.695, 75.883]
  MoveL 9058 to (-6.05, 64.85, -12.5) mm, rotated rx 180 ry 0 rz 90 deg; joints [75.883, -17.655, 85.908, 0, 21.746, 75.883]
  Establecer velocidad (1000.0 mm/s)
  MoveL 9059 to (-6.05, 64.85, 10) mm, rotated rx 180 ry 0 rz 90 deg; joints [75.883, -18.813, 86.664, 0, 22.15, 75.883]
  Establecer velocidad (66.7 mm/s)
  MoveL 9060 to (-61.48, 35.21, 10) mm, rotated rx -180 ry 0 rz 90 deg; joints [74.4, -19.602, 89.939, 0, 19.664, 74.4]
  MoveL 9061 to (-61.48, 35.21, -12.25) mm, rotated rx 180 ry 0 rz 90 deg; joints [74.4, -18.44, 89.191, 0, 19.248, 74.4]
  MoveL 9062 to (-62.98, 35.39, -12.66) mm, rotated rx -180 ry 0 rz 90 deg; joints [74.392, -18.442, 89.282, 0, 19.16, 74.392]
  MoveL 9063 to (-64.49, 35.21, -13.06) mm, rotated rx -180 ry 0 rz 90 deg; joints [74.372, -18.442, 89.367, 0, 19.076, 74.372]
  MoveL 9064 to (-65.92, 34.7, -13.47) mm, rotated rx 180 ry 0 rz 90 deg; joints [74.341, -18.44, 89.439, 0, 19.001, 74.341]
  MoveL 9065 to (-67.2, 33.88, -13.88) mm, rotated rx -180 ry 0 rz 90 deg; joints [74.301, -18.435, 89.496, 0, 18.939, 74.301]
  MoveL 9066 to (-68.27, 32.8, -14.28) mm, rotated rx 180 ry 0 rz 90 deg; joints [74.254, -18.425, 89.533, 0, 18.891, 74.254]
  MoveL 9067 to (-69.08, 31.51, -14.69) mm, rotated rx -180 ry 0 rz 90 deg; joints [74.203, -18.41, 89.549, 0, 18.861, 74.203]
  MoveL 9068 to (-69.58, 30.08, -15.09) mm, rotated rx 180 ry 0 rz 90 deg; joints [74.15, -18.39, 89.541, 0, 18.849, 74.15]
  MoveL 9069 to (-69.72, 28.57, -15.5) mm, rotated rx -180 ry 0 rz 90 deg; joints [74.097, -18.365, 89.508, 0, 18.857, 74.097]
  MoveL 9070 to (-69.72, 6.16, -15.5) mm, rotated rx 180 ry 0 rz 90 deg; joints [73.341, -18.267, 89.069, 0, 19.198, 73.341]
  MoveL 9071 to (-69.71, 5.21, -15.5) mm, rotated rx -180 ry 0 rz 90 deg; joints [73.309, -18.263, 89.05, 0, 19.213, 73.309]
  MoveC 9072 to (-68.74, 3.46, -15.5) mm, rotated rx 180 ry 0 rz 90 deg; joints [73.26, -18.241, 88.949, 0, 19.291, 73.26] to (-66.81, 2.92, -15.5) mm, rotated rx 180 ry 0 rz 90 deg; joints [73.262, -18.209, 88.809, 0, 19.4, 73.262]
  MoveC 9073 to (-46.96, 7.79, -15.5) mm, rotated rx 180 ry 0 rz 90 deg; joints [73.621, -17.923, 87.563, 0, 20.36, 73.621] to (-27.14, 12.79, -15.5) mm, rotated rx -180 ry 0 rz 90 deg; joints [73.977, -17.621, 86.3, 0, 21.322, 73.977]
  MoveL 9074 to (-27.01, 12.83, -15.5) mm, rotated rx -180 ry 0 rz 90 deg; joints [73.979, -17.619, 86.291, 0, 21.328, 73.979]
  MoveL 9075 to (-26.35, 13.05, -15.5) mm, rotated rx 180 ry 0 rz 90 deg; joints [73.993, -17.609, 86.25, 0, 21.359, 73.993]
  MoveC 9076 to (-25.03, 14.57, -15.5) mm, rotated rx 180 ry 0 rz 90 deg; joints [74.055, -17.594, 86.188, 0, 21.406, 74.055] to (-24.99, 16.58, -15.5) mm, rotated rx -180 ry 0 rz 90 deg; joints [74.122, -17.603, 86.226, 0, 21.378, 74.122]
  MoveL 9077 to (-29.34, 29.04, -15.5) mm, rotated rx -180 ry 0 rz 90 deg; joints [74.493, -17.735, 86.77, 0, 20.965, 74.493]
  MoveC 9078 to (-29.77, 29.82, -15.5) mm, rotated rx 180 ry 0 rz 90 deg; joints [74.515, -17.745, 86.814, 0, 20.931, 74.515] to (-30.42, 30.43, -15.5) mm, rotated rx 180 ry 0 rz 90 deg; joints [74.529, -17.759, 86.871, 0, 20.888, 74.529]
  MoveC 9079 to (-48.17, 42.27, -15.5) mm, rotated rx -180 ry 0 rz 90 deg; joints [74.762, -18.096, 88.311, 0, 19.785, 74.762] to (-65.99, 54.02, -15.5) mm, rotated rx -180 ry 0 rz 90 deg; joints [74.997, -18.413, 89.73, 0, 18.683, 74.997]
  MoveC 9080 to (-68.01, 53.9, -15.5) mm, rotated rx 180 ry 0 rz 90 deg; joints [74.974, -18.442, 89.863, 0, 18.579, 74.974] to (-69.54, 52.58, -15.5) mm, rotated rx -180 ry 0 rz 90 deg; joints [74.915, -18.459, 89.942, 0, 18.517, 74.915]
  MoveC 9081 to (-69.67, 52.26, -15.5) mm, rotated rx -180 ry 0 rz 90 deg; joints [74.903, -18.46, 89.945, 0, 18.515, 74.903] to (-69.72, 51.92, -15.5) mm, rotated rx 180 ry 0 rz 90 deg; joints [74.891, -18.459, 89.942, 0, 18.517, 74.891]
  MoveL 9082 to (-69.72, 28.57, -15.5) mm, rotated rx -180 ry 0 rz 90 deg; joints [74.097, -18.365, 89.508, 0, 18.857, 74.097]
  MoveL 9083 to (-62.16, 28.57, -15.5) mm, rotated rx -180 ry 0 rz 90 deg; joints [74.17, -18.252, 89.001, 0, 19.252, 74.17]
  MoveL 9084 to (-62.16, 28.57, -12.5) mm, rotated rx -180 ry 0 rz 90 deg; joints [74.17, -18.409, 89.103, 0, 19.306, 74.17]
  Establecer velocidad (1000.0 mm/s)
  MoveL 9085 to (-62.16, 28.57, 10) mm, rotated rx -180 ry 0 rz 90 deg; joints [74.17, -19.584, 89.859, 0, 19.725, 74.17]
  Establecer velocidad (66.7 mm/s)
  MoveL 9086 to (-40.12, -35.95, 10) mm, rotated rx 180 ry 0 rz 90 deg; joints [72.251, -18.906, 87.033, 0, 21.873, 72.251]
  MoveL 9087 to (-40.12, -35.95, -12.25) mm, rotated rx -180 ry 0 rz 90 deg; joints [72.251, -17.758, 86.286, 0, 21.473, 72.251]
  MoveL 9088 to (-40.23, -34.44, -12.66) mm, rotated rx -180 ry 0 rz 90 deg; joints [72.299, -17.747, 86.313, 0, 21.435, 72.299]
  MoveL 9089 to (-40.7, -33, -13.06) mm, rotated rx 180 ry 0 rz 90 deg; joints [72.341, -17.742, 86.363, 0, 21.379, 72.341]
  MoveL 9090 to (-41.48, -31.69, -13.47) mm, rotated rx 180 ry 0 rz 90 deg; joints [72.375, -17.741, 86.431, 0, 21.31, 72.375]
  MoveL 9091 to (-42.52, -30.59, -13.88) mm, rotated rx 180 ry 0 rz 90 deg; joints [72.401, -17.743, 86.513, 0, 21.231, 72.401]
  MoveL 9092 to (-43.79, -29.75, -14.28) mm, rotated rx 180 ry 0 rz 90 deg; joints [72.415, -17.748, 86.604, 0, 21.144, 72.415]
  MoveL 9093 to (-45.21, -29.21, -14.69) mm, rotated rx -180 ry 0 rz 90 deg; joints [72.418, -17.753, 86.699, 0, 21.054, 72.418]
  MoveL 9094 to (-46.72, -28.99, -15.09) mm, rotated rx 180 ry 0 rz 90 deg; joints [72.409, -17.758, 86.793, 0, 20.965, 72.409]
  MoveL 9095 to (-48.22, -29.15, -15.5) mm, rotated rx -180 ry 0 rz 90 deg; joints [72.389, -17.761, 86.878, 0, 20.882, 72.389]
  MoveL 9096 to (-64.91, -32.42, -15.5) mm, rotated rx 180 ry 0 rz 90 deg; joints [72.105, -18.011, 87.94, 0, 20.071, 72.105]
  MoveL 9097 to (-67.73, -32.98, -15.5) mm, rotated rx 180 ry 0 rz 90 deg; joints [72.056, -18.052, 88.117, 0, 19.934, 72.056]
  MoveC 9098 to (-69.11, -33.79, -15.5) mm, rotated rx -180 ry 0 rz 90 deg; joints [72.015, -18.069, 88.192, 0, 19.877, 72.015] to (-69.7, -35.28, -15.5) mm, rotated rx -180 ry 0 rz 90 deg; joints [71.959, -18.07, 88.199, 0, 19.871, 71.959]
  MoveL 9099 to (-69.71, -35.54, -15.5) mm, rotated rx 180 ry 0 rz 90 deg; joints [71.95, -18.069, 88.195, 0, 19.875, 71.95]
  MoveL 9100 to (-69.71, -67.07, -15.5) mm, rotated rx -180 ry 0 rz 90 deg; joints [70.913, -17.904, 87.482, 0, 20.422, 70.913]
  MoveC 9101 to (-68.96, -68.87, -15.5) mm, rotated rx 180 ry 0 rz 90 deg; joints [70.863, -17.882, 87.39, 0, 20.492, 70.863] to (-67.15, -69.59, -15.5) mm, rotated rx -180 ry 0 rz 90 deg; joints [70.86, -17.849, 87.251, 0, 20.598, 70.86]
  MoveC 9102 to (-52.66, -69.26, -15.5) mm, rotated rx 180 ry 0 rz 90 deg; joints [71.033, -17.615, 86.276, 0, 21.339, 71.033] to (-38.17, -68.87, -15.5) mm, rotated rx 180 ry 0 rz 90 deg; joints [71.206, -17.372, 85.291, 0, 22.081, 71.206]
  MoveC 9103 to (-36.6, -68.29, -15.5) mm, rotated rx -180 ry 0 rz 90 deg; joints [71.241, -17.349, 85.196, 0, 22.152, 71.241] to (-35.69, -66.88, -15.5) mm, rotated rx 180 ry 0 rz 90 deg; joints [71.296, -17.341, 85.167, 0, 22.175, 71.296]
